// TwinCAT 3 PLC project SPT_PackML_Base
// Title: SPT PackML Base
// Company: Beckhoff Automation LLC
// ProjectVersion: 4.0.0.0
// Description: 4.0.0.0 - Bonkers
// libraries:
//   Intecre.Utilities, * (Intecre Ltd)
//   SPT Event Logger, * (Beckhoff Automation LLC)
//   SPT Utilities, * (Beckhoff Automation LLC)
//   Tc2_Standard, * (Beckhoff Automation GmbH)
//   Tc2_System, * (Beckhoff Automation GmbH)
//   Tc3_EventLogger, * (Beckhoff Automation GmbH)
//   Tc3_Module, * (Beckhoff Automation GmbH)
//   Tc3_PackML_V2, * (Beckhoff Automation GmbH)
//   tcl_SimpleUnitTestLibrary, * (Red Rock Controls Limited)
//   SPT Base Types,newest,Beckhoff Automation LLC
//   SPT Component Base,newest,Beckhoff Automation LLC
// project tree:
//   DUT/ E_PMLUnitMode.TcDUT, ST_PackML_SubUnitInfoExt.TcDUT
//   DUT/HMI/ ST_PackMLBaseModule_Command.TcDUT, ST_PackMLBaseModule_Config.TcDUT, ST_PackMLBaseModule_HMI.TcDUT, ST_PackMLBaseModule_Status.TcDUT
//   Example things/ I_ExampleEquipment.TcIO, T_ExampleModule.TcPOU, T_ExampleMOduleProductionMode.TcPOU
//   / FB_PackML_BaseModule.TcPOU, FB_PackML_ModeLogger.TcPOU, FB_PackML_StateLogger.TcPOU, GlobalTextList.TcGTLO, Parameters_PackML_Base.TcGVL, Task_3.TcTTO, TestUI.TcVIS, Visualization Manager.TcVMO (not stored)
//   Intecre/Axis/ I_Axis.TcIO, I_AxisComponent.TcIO, T_Axis.TcPOU, T_AxisComponent.TcPOU
//   Intecre/CartesianRobot/ I_CartesianRobot.TcIO, I_CartesianRobotModule.TcIO, T_CartesianRobotModule.TcPOU, T_CartesianRobot.TcPOU
//   Intecre/CartesianRobot/Modes/ T_CartesianRobotMaintenanceMode.TcPOU, T_CartesianRobotManualMode.TcPOU, T_CartesianRobotProductionMode.TcPOU
//   Intecre/Collections/ I_ComponentsCollection.TcIO, I_SubModuleCollection.TcIO, T_BaseAlarms.TcPOU, T_CollectionBase.TcPOU, T_ComponentsCollection.TcPOU, T_ExternalControllerCollection.TcPOU, T_SubModuleCollection.TcPOU
//   Intecre/Gripper/ I_Gripper.TcIO, I_GripperModule.TcIO, T_Gripper.TcPOU, T_GripperModule.TcPOU
//   Intecre/Gripper/Modes/ T_GripperMaintenanceMode.TcPOU, T_GripperManualMode.TcPOU, T_GripperProductionMode.TcPOU
//   Intecre/ModeManager/ I_ModeManager.TcIO, T_ModeManager.TcPOU
//   Intecre/PackModes/ I_PackMode.TcIO, I_StateModule.TcIO, T_BaseMode.TcPOU
//   Intecre/Cylinder/ I_Cylinder.TcIO, I_CylinderComponent.TcIO, T_Cylinder.TcPOU, T_CylinderComponent.TcPOU
//   Interfaces/ I_PackML_BaseModule.TcIO, I_PackML_Control.TcIO, I_PackML_ExternalController.TcIO
//   Project Information/ F_GetCompany.TcPOU, F_GetTitle.TcPOU, F_GetVersion.TcPOU
//   Tests/AlarmsTests/ T_BaseAlarmsClearAlarmIfRaisedCleared.TcPOU
//   Tests/CollectionsTests/Components/Mock/ T_ComponentMock.TcPOU (not stored)
//   Tests/CollectionsTests/Components/ T_AddComponentAddedToList.TcPOU, T_AddComponentCompareResultTrue.TcPOU, T_AddMoreThanSizeOfCollectionFalse.TcPOU, T_AddSameComponentTwiceShouldntAdd.TcPOU, T_ClearGroupCountEqualsZeroCompareEqualsFalse.TcPOU, T_ComponentsAllowHmiAllowed.TcPOU, T_ComponentsBlockHmiBlocked.TcPOU (not stored), T_ComponentsIfAnyErrorReturnsErrorTrue.TcPOU (not stored), T_ComponentsInitialisedSuccess.TcPOU (not stored), T_ComponentsResetClearsErrors.TcPOU (not stored), T_CountReturnsCorrect.TcPOU, T_CyclicLogicHasBeenCalledTrue.TcPOU (not stored), T_GetComponentCompareResultsTrue.TcPOU (not stored), T_GetComponentIndexOutOfBoundaryResultsFalse.TcPOU
//   Tests/CollectionsTests/ExternalController/Mock/ T_ExternalControllerMock.TcPOU (not stored)
//   Tests/CollectionsTests/ExternalController/ T_ExternalControllersCollectionNotifyModeChangedSuccess.TcPOU (not stored), T_ExternalControllersCollectionNotifyStateChangedSuccess.TcPOU (not stored)
//   Tests/CollectionsTests/Module/Mock/ T_SubModuleMock.TcPOU (not stored)
//   Tests/CollectionsTests/Module/ T_ModuleCollectionAllInAskedStateReturnsCorrectResponse.TcPOU, T_ModuleCollectionAnyErrorReturnErrorTrue.TcPOU, T_ModuleCollectionAnyInAskedStateReturnsCorrectResponse.TcPOU, T_ModuleCollectionInitialisedSuccess.TcPOU (not stored), T_ModuleCollectionNotifyModeChangedSuccess.TcPOU (not stored), T_ModuleCollectionNotifyStateChangedSuccess.TcPOU (not stored), T_ModuleCollectionOneIsNotInAskedStateReturnsCorrectResponse.TcPOU, T_ModuleCollectionOneNotInitialisedAllNotInitialised.TcPOU, T_ModuleCollectionStateResetReturnsCorrectResponse.TcPOU
//   Tests/ModeAndStateTests/ EquipmentModule.TcPOU, T_CantChangeModInExecute.TcPOU, T_CantChangeStateFromIdleToSuspend.TcPOU, T_JogThroughStates.TcPOU, T_ProductionToMaintenaceInAbort.TcPOU
//   Tests/ModeManagerTests/Mock Objects/ T_MockStateModule.TcPOU
//   Tests/ModeManagerTests/ T_AddCustomPackModeSetsCorrectly.TcPOU, T_AddPackModeSetsCorrectly.TcPOU, T_InitModeManagerWithState.TcPOU, T_ModeChangeFromProductionToMaintenance.TcPOU, T_ModeInitialisedFromInvalidToProduction.TcPOU
//   Tests/ PRG_Tests.TcPOU
//   Version/ Global_Version.TcGVL
//   VISUs/ V_MachineModule.TcVIS, V_Module.TcVIS
// (motion and I/O tree: see PLC project spt_base_types)
// real-time tasks:
//   TASK Task 3: cycle T#10ms, priority 1, ADS port 350

CONFIGURATION SPT_PackML_Base
    RESOURCE PLC ON TwinCAT3
        TASK Task_3(INTERVAL := T#10ms, PRIORITY := 1);
        PROGRAM PRG_Tests WITH Task_3 : PRG_Tests;
    END_RESOURCE
END_CONFIGURATION

// ---- DUT/E_PMLUnitMode.TcDUT
//! @summary Defines the allowable PackML modes  
TYPE E_PMLUnitMode : (
        ePMLUnitMode_Invalid     := 0,
        ePMLUnitMode_Production  := 1,
        ePMLUnitMode_Maintenance := 2,
        ePMLUnitMode_Manual      := 3,
        ePMLUnitMode_UserMode1   := 4,
        ePMLUnitMode_UserMode2   := 5,
        ePMLUnitMode_UserMode3   := 6,
        ePMLUnitMode_UserMode4   := 7,
        ePMLUnitMode_UserMode5   := 8,
        ePMLUnitMode_UserMode6   := 9,
        ePMLUnitMode_UserMode7   := 10,
        ePMLUnitMode_UserMode8   := 11,
        ePMLUnitMode_UserMode9   := 12,
        ePMLUnitMode_UserMode10  := 13,
        ePMLUnitMode_UserMode11  := 14,
        ePMLUnitMode_UserMode12  := 15,
        ePMLUnitMode_UserMode13  := 16,
        ePMLUnitMode_UserMode14  := 17,
        ePMLUnitMode_UserMode15  := 18,
        ePMLUnitMode_UserMode16  := 19,
        ePMLUnitMode_UserMode17  := 20,
        ePMLUnitMode_UserMode18  := 21,
        ePMLUnitMode_UserMode19  := 22,
        ePMLUnitMode_UserMode20  := 23,
        ePMLUnitMode_UserMode21  := 24,
        ePMLUnitMode_UserMode22  := 25,
        ePMLUnitMode_UserMode23  := 26,
        ePMLUnitMode_UserMode24  := 27,
        ePMLUnitMode_UserMode25  := 28,
        ePMLUnitMode_UserMode26  := 29,
        ePMLUnitMode_UserMode27  := 30,
        ePMLUnitMode_UserMode28  := 31
    ) DINT;
END_TYPE

// ---- DUT/HMI/ST_PackMLBaseModule_Command.TcDUT
TYPE ST_PackMLBaseModule_Command :
    STRUCT
        Mode               : E_PMLUnitMode              := Parameters_PackML_Base.UNIT_MODE_DEFAULT;
        State              : Tc3_PackML_V2.E_PMLCommand := Parameters_PackML_Base.UNIT_STATE_DEFAULT;
        ActivateStateLog   : BOOL; //HMI requests to enable the module
        DeactivateStateLog : BOOL; //HMI requests to disable the module
        ActivateModeLog    : BOOL; //HMI requests to enable the module
        DeactivatModeLog   : BOOL; //HMI requests to disable the module
    END_STRUCT
END_TYPE

// ---- DUT/HMI/ST_PackMLBaseModule_Config.TcDUT
TYPE ST_PackMLBaseModule_Config :
    STRUCT
        Name            : STRING;       //Human-readable module name for user-side messaging
        LogStateChanges : BOOL := TRUE; //Toggle to permit or suppress state change logging (Should be tied to HMI setting to optionally reduce event logger clutter)
        LogModeChanges  : BOOL := TRUE; //Toggle to permit or suppress state change logging (Should be tied to HMI setting to optionally reduce event logger clutter)
        ModeNames       : ARRAY[0..31] OF STRING;
    END_STRUCT
END_TYPE

// ---- DUT/HMI/ST_PackMLBaseModule_HMI.TcDUT
TYPE ST_PackMLBaseModule_HMI :
    STRUCT
        Config  : ST_PackMLBaseModule_Config;
        Command : ST_PackMLBaseModule_Command;
        Status  : ST_PackMLBaseModule_Status;
    END_STRUCT
END_TYPE

// ---- DUT/HMI/ST_PackMLBaseModule_Status.TcDUT
TYPE ST_PackMLBaseModule_Status :
    STRUCT
        Busy                : BOOL;
        Error               : BOOL;
        ErrorID             : UDINT;
        Mode                : E_PMLUnitMode;
        State               : Tc3_PackML_V2.E_PMLState;
        HMIControlAvailable : BOOL;
    END_STRUCT
END_TYPE

// ---- DUT/ST_PackML_SubUnitInfoExt.TcDUT
TYPE ST_PackML_SubUnitInfoExt EXTENDS ST_PMLSubUnitInfo : //Extended Struct of ST_PMLSubUnitInfo
    STRUCT
        ModuleID        : DINT;   //Machine ID for messaging and Identification
        ModuleName      : STRING; //Human readable machine name for messaging
        UnitModeCurrent : E_PMLProtectedUnitMode;
        ActiveAlarm     : BOOL;
    END_STRUCT
END_TYPE

// ---- Parameters_PackML_Base.TcGVL
{attribute 'qualified_only'}
VAR_GLOBAL CONSTANT
    MAX_NO_OF_SUBMODULES           : UDINT                       := 20;
    MAX_NO_OF_COMPONENTS           : UDINT                       := 32;
    MAX_NO_OF_EXTERNAL_CONTROLLERS : UDINT                       := 10;
    UNIT_MODE_DEFAULT              : E_PMLUnitMode := E_PMLUnitMode.ePMLUnitMode_Production;
    UNIT_STATE_DEFAULT             : Tc3_PackML_V2.E_PMLCommand  := E_PMLCommand.ePMLCommand_Abort;
	COLLECTION_MAX_SIZE : UDINT := 200;
END_VAR

// ---- Version/Global_Version.TcGVL
{attribute 'TcGenerated'}
{attribute 'no-analysis'}
{attribute 'linkalways'}
// This function has been automatically generated from the project information.
VAR_GLOBAL CONSTANT
	{attribute 'const_non_replaced'}
	stLibVersion_SPT_PackML_Base : ST_LibVersion := (iMajor := 3, iMinor := 0, iBuild := 3, iRevision := 0, nFlags := 1, sVersion := '3.0.3');
END_VAR

// ---- Example things/I_ExampleEquipment.TcIO
INTERFACE I_ExampleEquipment EXTENDS I_PackML_BaseModule

METHOD PUBLIC PickFromStagingArea : BOOL
VAR_INPUT
  orientationOfPick : ST_Orientation;
END_VAR
END_METHOD

END_INTERFACE

// ---- Intecre/Axis/I_Axis.TcIO
INTERFACE I_Axis

END_INTERFACE

// ---- Intecre/Axis/I_AxisComponent.TcIO
INTERFACE I_AxisComponent

END_INTERFACE

// ---- Intecre/CartesianRobot/I_CartesianRobot.TcIO
INTERFACE I_CartesianRobot

METHOD GenericInitialise : BOOL;
VAR_INPUT
	xAxis, yAxis, zAxis : I_Axis;
	gripper : I_Gripper;
END_VAR
END_METHOD

END_INTERFACE

// ---- Intecre/CartesianRobot/I_CartesianRobotModule.TcIO
INTERFACE I_CartesianRobotModule

END_INTERFACE

// ---- Intecre/Collections/I_ComponentsCollection.TcIO
INTERFACE I_ComponentsCollection

END_INTERFACE

// ---- Intecre/Collections/I_SubModuleCollection.TcIO
INTERFACE I_SubModuleCollection

PROPERTY Count : UDINT
GET
END_GET
END_PROPERTY

METHOD TryGetModule: BOOL
VAR_INPUT
	index : UDINT;
END_VAR
VAR_OUTPUT
	Module : I_PackML_BaseModule;
END_VAR
END_METHOD

END_INTERFACE

// ---- Intecre/Gripper/I_Gripper.TcIO
INTERFACE I_Gripper

END_INTERFACE

// ---- Intecre/Gripper/I_GripperModule.TcIO
INTERFACE I_GripperModule

END_INTERFACE

// ---- Intecre/ModeManager/I_ModeManager.TcIO
INTERFACE I_ModeManager

METHOD AddCustomPackMode : BOOL
VAR_INPUT
  index : UINT;
  newPackMode : I_PackMode;
END_VAR
END_METHOD

METHOD AddPackModes : BOOL
VAR_INPUT
  prodMode : I_PackMode;
  maintMode : I_PackMode;
  manMode : I_PackMode;
END_VAR
END_METHOD

METHOD PUBLIC AddStateModule
VAR_INPUT
  stateModule : I_StateModule;
END_VAR
END_METHOD

METHOD PUBLIC ChangeMode
VAR_INPUT
  Mode : E_PMLUnitMode;
END_VAR
END_METHOD

PROPERTY PUBLIC CommandedMode : E_PMLUnitMode
GET
END_GET
END_PROPERTY

PROPERTY CurrentMode : E_PMLUnitMode
GET
END_GET
END_PROPERTY

METHOD PUBLIC CyclicLogic
VAR_INPUT
END_VAR
END_METHOD

PROPERTY PUBLIC LogModeChanges : BOOL
GET
END_GET
SET
END_SET
END_PROPERTY

PROPERTY PUBLIC  ModeNames : REFERENCE TO ARRAY[0..31] OF STRING
GET
END_GET
END_PROPERTY

END_INTERFACE

// ---- Intecre/PackModes/I_PackMode.TcIO
INTERFACE I_PackMode

METHOD Aborted
VAR_INPUT
END_VAR
END_METHOD

METHOD Aborting
VAR_INPUT
END_VAR
END_METHOD

METHOD Clearing
VAR_INPUT
END_VAR
END_METHOD

METHOD Complete
VAR_INPUT
END_VAR
END_METHOD

METHOD Completing
VAR_INPUT
END_VAR
END_METHOD

METHOD Execute
VAR_INPUT
END_VAR
END_METHOD

METHOD Held
VAR_INPUT
END_VAR
END_METHOD

METHOD Holding
VAR_INPUT
END_VAR
END_METHOD

METHOD Idle
VAR_INPUT
END_VAR
END_METHOD

METHOD Resetting
VAR_INPUT
END_VAR
END_METHOD

METHOD Starting
VAR_INPUT
END_VAR
END_METHOD

METHOD Stopped
VAR_INPUT
END_VAR
END_METHOD

METHOD Stopping
VAR_INPUT
END_VAR
END_METHOD

METHOD Suspended
VAR_INPUT
END_VAR
END_METHOD

METHOD Suspending
VAR_INPUT
END_VAR
END_METHOD

METHOD Unholding
VAR_INPUT
END_VAR
END_METHOD

METHOD Unsuspending
VAR_INPUT
END_VAR
END_METHOD

END_INTERFACE

// ---- Intecre/PackModes/I_StateModule.TcIO
INTERFACE I_StateModule

PROPERTY CurrentState : Tc3_PackML_V2.E_PMLState
GET
END_GET
END_PROPERTY

END_INTERFACE

// ---- Intecre/Cylinder/I_Cylinder.TcIO
INTERFACE I_Cylinder

END_INTERFACE

// ---- Intecre/Cylinder/I_CylinderComponent.TcIO
INTERFACE I_CylinderComponent

END_INTERFACE

// ---- Interfaces/I_PackML_BaseModule.TcIO
INTERFACE I_PackML_BaseModule EXTENDS I_CyclicFB, I_PackML_Control

PROPERTY CurrentAlarmSeverity : TcEventSeverity
GET
END_GET
END_PROPERTY

PROPERTY LogModeChanges : BOOL
GET
END_GET
SET
END_SET
END_PROPERTY

PROPERTY LogStateChanges : BOOL
GET
END_GET
SET
END_SET
END_PROPERTY

PROPERTY Name : STRING
GET
END_GET
SET
END_SET
END_PROPERTY

PROPERTY ParentResponseDefinitions : ARRAY[0..4] OF E_AlarmResponse
GET
END_GET
SET
END_SET
END_PROPERTY

END_INTERFACE

// ---- Interfaces/I_PackML_Control.TcIO
INTERFACE I_PackML_Control EXTENDS I_InterfaceBase

METHOD ChangeMode
VAR_INPUT
    Mode : E_PMLUnitMode;
END_VAR
END_METHOD

METHOD ChangeState
VAR_INPUT
    State : E_PMLCommand;
END_VAR
END_METHOD

PROPERTY CurrentMode : E_PMLUnitMode
GET
END_GET
END_PROPERTY

PROPERTY CurrentState : E_PMLState
GET
END_GET
END_PROPERTY

PROPERTY ModeCommand : DINT
GET
END_GET
SET
END_SET
END_PROPERTY

PROPERTY StateCommand : E_PMLCommand
GET
END_GET
SET
END_SET
END_PROPERTY

END_INTERFACE

// ---- Interfaces/I_PackML_ExternalController.TcIO
INTERFACE I_PackML_ExternalController EXTENDS I_InterfaceBase

PROPERTY Control : I_PackML_Control
SET
END_SET
END_PROPERTY

METHOD ModeChanged
VAR_INPUT
    NewMode : E_PMLUnitMode;
END_VAR
END_METHOD

METHOD StateChanged
VAR_INPUT
    NewState : E_PMLCommand;
END_VAR
END_METHOD

END_INTERFACE

// ---- Tests/PRG_Tests.TcPOU
PROGRAM PRG_Tests
VAR
  testRunner : T_TestRunner;
  
  //Modes
  modeTestSuite : T_TestSuite;
  ProductionToMaintenaceInAbort : T_ProductionToMaintenaceInAbort(modeTestSuite);
  CantChangeModInExecute : T_CantChangeModInExecute(modeTestSuite);
  JogThroughStates : T_JogThroughStates(modeTestSuite);
  CantChangeStateFromIdleToSuspend : T_CantChangeStateFromIdleToSuspend(modeTestSuite);
  
  // set mode
  AddPackModeSetsCorrectly : T_AddPackModeSetsCorrectly(modeTestSuite);  
  InitModeManagerWithState : T_InitModeManagerWithState(modeTestSuite);
  ModeChangeFromProductionToMaintenance : T_ModeChangeFromProductionToMaintenance(modeTestSuite);
  ModeInitialisedFromInvalidToProduction : T_ModeInitialisedFromInvalidToProduction(modeTestSuite);
  AddCustomPackModeSetsCorrectly : T_AddCustomPackModeSetsCorrectly(modeTestSuite);
  
    //collections tests
  CollectionsTestSuite : T_TestSuite;
  AddComponentAddedToList : T_AddComponentAddedToList (CollectionsTestSuite);
  AddComponentCompareResultTrue : T_AddComponentCompareResultTrue(CollectionsTestSuite);
  CountReturnsCorrect : T_CountReturnsCorrect(CollectionsTestSuite);
  GetComponentCompareResultsTrue : T_GetComponentCompareResultsTrue(CollectionsTestSuite);
  ClearGroupCountEqualsZeroCompareEqualsFalse : T_ClearGroupCountEqualsZeroCompareEqualsFalse(CollectionsTestSuite);
  AddSameComponentTwiceShouldntAdd : T_AddSameComponentTwiceShouldntAdd(CollectionsTestSuite);
  GetComponentIndexOutOfBoundaryResultsFalse : T_GetComponentIndexOutOfBoundaryResultsFalse(CollectionsTestSuite);
  AddMoreThanSizeOfCollectionFalse : T_AddMoreThanSizeOfCollectionFalse(CollectionsTestSuite);
  CyclicLogicHasBeenCalledTrue : T_CyclicLogicHasBeenCalledTrue(CollectionsTestSuite);
  ComponentsInitialisedSuccess : T_ComponentsInitialisedSuccess (CollectionsTestSuite);
  ComponentsIfAnyErrorReturnsErrorTrue : T_ComponentsIfAnyErrorReturnsErrorTrue (CollectionsTestSuite);
  ComponentsAllowHmiAllowed : T_ComponentsAllowHmiAllowed (CollectionsTestSuite);
  ComponentsBlockHmiBlocked : T_ComponentsBlockHmiBlocked (CollectionsTestSuite);
  ComponentsResetClearsErrors : T_ComponentsResetClearsErrors (CollectionsTestSuite);
  ExternalControllersCollectionNotifyStateChangedSuccess : T_ExternalControllersCollectionNotifyStateChangedSuccess (CollectionsTestSuite);
  ExternalControllersCollectionNotifyModeChangedSuccess : T_ExternalControllersCollectionNotifyModeChangedSuccess (CollectionsTestSuite);
  ModuleCollectionNotifyModeChangedSuccess : T_ModuleCollectionNotifyModeChangedSuccess (CollectionsTestSuite);
  ModuleCollectionNotifyStateChangedSuccess : T_ModuleCollectionNotifyStateChangedSuccess (CollectionsTestSuite);
  ModuleCollectionInitialisedSuccess : T_ModuleCollectionInitialisedSuccess (CollectionsTestSuite);
  ModuleCollectionOneNotInitialisedAllNotInitialised : T_ModuleCollectionOneNotInitialisedAllNotInitialised (CollectionsTestSuite);
  ModuleCollectionAnyErrorReturnErrorTrue : T_ModuleCollectionAnyErrorReturnErrorTrue (CollectionsTestSuite);
  ModuleCollectionAllInAskedStateReturnsCorrectResponse : T_ModuleCollectionAllInAskedStateReturnsCorrectResponse (CollectionsTestSuite);
  ModuleCollectionOneIsNotInAskedStateReturnsCorrectResponse : T_ModuleCollectionOneIsNotInAskedStateReturnsCorrectResponse (CollectionsTestSuite);
  ModuleCollectionAnyInAskedStateReturnsCorrectResponse : T_ModuleCollectionAnyInAskedStateReturnsCorrectResponse (CollectionsTestSuite);
  ModuleCollectionStateResetReturnsCorrectResponse : T_ModuleCollectionStateResetReturnsCorrectResponse (CollectionsTestSuite);
END_VAR

IF testRunner.ReloadTests THEN
    testRunner.AddTestSuite(modeTestSuite);
    testRunner.AddTestSuite(CollectionsTestSuite);
    testRunner.ReloadTests := FALSE;
END_IF

testRunner();

END_PROGRAM

// ---- Tests/ModeAndStateTests/T_ProductionToMaintenaceInAbort.TcPOU
FUNCTION_BLOCK T_ProductionToMaintenaceInAbort EXTENDS T_UnitTestBase
VAR
  em : EquipmentModule; 
  actual, expected : E_PMLUnitMode;
  scanCounter: INT;
  cmdTriggered : BOOL;
  myTestState : (ARRANGE, ACT, ASSERT);
END_VAR

CASE myTestState OF

  ARRANGE:
    em.CyclicLogic();

    IF em.InitComplete THEN
      myTestState := ACT;
      CycleModuleLogicToAllowChangesToFilterThrough();
    END_IF

  ACT:

    CycleModuleLogicToAllowChangesToFilterThrough();
    em.ChangeMode(E_PMLUnitMode.ePMLUnitMode_Maintenance);
    CycleModuleLogicToAllowChangesToFilterThrough();
    actual := em.CurrentMode;
    expected := E_PMLUnitMode.ePMLUnitMode_Maintenance;
    myTestState := ASSERT;

  ASSERT:

    assertion.AssertEquals_UINT(TO_UINT(actual), TO_UINT(expected), 'actual := equipmentModule.CurrentMode');
    myTestState := ARRANGE;
    cmdTriggered := FALSE;
    TestFinished();

END_CASE

METHOD CycleModuleLogicToAllowChangesToFilterThrough : BOOL
VAR_INST
	i: INT;

END_VAR
//em.CyclicLogic();
//CycleModuleLogicToAllowChangesToFilterThrough := i >= 10;
//i := SEL(i >= 10, i + 1, 0);

FOR i := 0 TO 10 DO
  em.CyclicLogic();
END_FOR
END_METHOD

END_FUNCTION_BLOCK

// ---- Tests/ModeAndStateTests/EquipmentModule.TcPOU
FUNCTION_BLOCK EquipmentModule EXTENDS FB_PackML_BaseModule
VAR_INPUT
END_VAR
VAR_OUTPUT
END_VAR
VAR
END_VAR

END_FUNCTION_BLOCK

// ---- FB_PackML_BaseModule.TcPOU
FUNCTION_BLOCK ABSTRACT FB_PackML_BaseModule EXTENDS FB_CyclicFB IMPLEMENTS I_PackML_BaseModule, I_PackML_Control, I_StateModule
  //I_PMLControl
VAR

  _CurrentState : Tc3_PackML_V2.E_PMLState;
  _CommandedState : Tc3_PackML_V2.E_PMLCommand;
END_VAR

VAR
  _CurrentAlarmSeverity : TcEventSeverity;
  _LogStateChanges : BOOL := FALSE; //Toggle to permit or suppress state change logging (Should be tied to HMI setting to optionally reduce event logger clutter)
  _Name : STRING; //Human-readable module name for user-side messaging
  _ParentFaultResponseDefinitions : ARRAY[0..4] OF E_AlarmResponse
    := [E_AlarmResponse.NoResponse,
    E_AlarmResponse.NoResponse, E_AlarmResponse.NoResponse, E_AlarmResponse.Abort_ImmediateError, E_AlarmResponse.Abort_ImmediateError];
END_VAR

VAR

  ModeManager : T_ModeManager(THIS^);
  InitialiseStates : (init,
    CountSubModules,
    SetSizeOfArrays,
    WaitForInitializeComplete);
  ComponentsCollection : T_ComponentsCollection;
  SubModulesCollection : T_SubModuleCollection;
  ExternalControllersCollection : T_ExternalControllerCollection;
  BaseAlarms : T_BaseAlarms;

  //spt classes    
  StateMachine : PML_StateMachine; //Manages PackML state transitions   
  PrevState : Tc3_PackML_V2.E_PMLState; //Last cycle PackML state 
  PMLStateLogger : FB_PackML_StateLogger; //Logs PackML state changes

  PackMLAlarms : ARRAY[1..48] OF FB_TcAlarm; //Array of alarms for PackML state and mode changes that exist in any PackML enabled module
  ipSubModules : ARRAY[1..Parameters_PackML_Base.MAX_NO_OF_SUBMODULES] OF I_PackML_BaseModule;
  NumberOfSubModules : UDINT := 0; //calculated number of instantiated sub modules
  ReachedInitialDefaultStateAndMode : BOOL;

  HMICommand_RT : R_TRIG;
  HMICommandActive_Base : BOOL;
  HMICommandActive_Descendant : BOOL;
  PackMLBaseModule_HMI : ST_PackMLBaseModule_HMI; //Handles status and control communications with the HMI
END_VAR

//*********************************************************

// !!!!! Code implementation only in CyclicLogic() method !!!!! 

//*********************************************************

//! @summary This method contains code which will execute when this PackML module is in the <b>Aborted</b> state
METHOD PROTECTED Aborted

(*! <description> <b>The base implementation of this method is empty. User must override this method to provide functionality.</b>
<table> 
	<tr>
		<th> Previous State </th>
		<th> Transition In </th>
		<th> Transition Out </th>
		<th> Next State  </th> 
	</tr>
	<tr>
		<td> Aborting </td>
		<td> State Complete <i>(Aborting)</i></td> 
		<td> Clear Command </td>
		<td> Clearing </td> 
	</tr>
</table>
This method is called as required by <c>StateControl()</c>
</description> 

*)
//*************************************************************************************************************************************************************************

//If you are about to write application specific code, note that any such code should exist within the "Application" directory using a Function Block that 'EXTENDS' this base Function Block!

//This particular method's functionality can be overriden in the extended block by creating a method of the same name, with desired functionality therein

//If the functionality of this base module is to be retained, but more functionality is desired, the extended method can contain a SUPER^.ThisMethodName(); call, which will call this code

//*************************************************************************************************************************************************************************
END_METHOD

//! @summary Provides fault reaction logic where the module state is driven to the <b>Aborting</b> state
METHOD PROTECTED AbortImmediate

//! @description No error is thrown by this fault reaction.

//! @description This method is called by <c>ComponentMonitor()</c> or <c>SubModuleMonitor()</c> as required
ChangeState(E_PMLCommand.ePMLCommand_Abort);
END_METHOD

//! @summary Provides fault reaction logic where the module state is driven to the <b>Aborting</b> state
METHOD PROTECTED AbortImmediateError
VAR_INPUT
    Name     : STRING; //! The name of the faulting submodule or component
    IsModule : BOOL;   //! If TRUE a SubModuleError is thrown.  If FALSE a ComponentError is thrown. 
END_VAR

//! @description This fault reaction throws an accompanying error

//! @description This method is called by <c>ComponentMonitor()</c> or <c>SubModuleMonitor()</c> as required
//IF IsModule THEN
//    IF NOT BaseAlarms[E_BaseAlarms.SubModuleError].bRaised THEN
//        F_RaiseAlarmWithStringParameters(BaseAlarms[E_BaseAlarms.SubModuleError],
//                                         _Name,
//                                         '',
//                                         '');
//    END_IF
//ELSE
//    IF NOT BaseAlarms[E_BaseAlarms.ComponentError].bRaised THEN
//        F_RaiseAlarmWithStringParameters(BaseAlarms[E_BaseAlarms.ComponentError],
//                                         _Name,
//                                         '',
//                                         '');
//    END_IF
//END_IF

IF IsModule THEN
	BaseAlarms.RaiseAlarmWithStringParameters(E_BaseAlarms.SubModuleError, _name, '','');
ELSE
	BaseAlarms.RaiseAlarmWithStringParameters(E_BaseAlarms.ComponentError, _name, '','');
END_IF

THIS^.ChangeState(E_PMLCommand.ePMLCommand_Abort);
END_METHOD

//! @summary This method contains code which will execute when this PackML module is in the <b>Aborting</b> state
METHOD PROTECTED Aborting
(*! <description> <b>Note:</b> The <i>Abort</i> command should be associated with the fault handing routine of a module. It should not be directly commanded from any user inteface. 

<table> 
	<tr>
		<th> Previous State </th>
		<th> Transition In </th>
		<th> Transition Out </th>
		<th> Next State  </th> 
	</tr>
	<tr>
		<td> <b>ANY</b> </td>
		<td> Abort Command </td> 
		<td> State Complete </td>
		<td> Aborted </td> 
	</tr>
</table>

This method is called as required by <c>StateControl()</c>
</description> 

*)
//*************************************************************************************************************************************************************************

//If you are about to write application specific code, note that any such code should exist within the "Application" directory using a Function Block that 'EXTENDS' this base Function Block!

//This particular method's functionality can be overriden in the extended block by creating a method of the same name, with desired functionality therein

//If the functionality of this base module is to be retained, but more functionality is desired, the extended method can contain a SUPER^.ThisMethodName(); call, which will call this code

//*************************************************************************************************************************************************************************

//Perform State tasks here

// Send abort command to all sub modules
SubModulesCollection.NotifyStateChanged(ePMLCommand_Abort);

IF NOT SubModulesCollection.AllInRequestedState(ePMLState_Aborted) THEN
	RETURN;
END_IF

StateComplete();
END_METHOD

//! @summary Sets permissive bit to allow HMI control of module and component functions
METHOD PROTECTED FINAL AllowHMIControl
VAR_INPUT
    ThisModuleOnly : BOOL; //! If TRUE, only the PackML module itself is controllable. If FALSE, all components become controllable as well
END_VAR

VAR
    i : UDINT;
END_VAR

//! @description This method is called as required by the <c>HMIPermissions()</c> method
PackMLBaseModule_HMI.Status.HMIControlAvailable := TRUE;
IF ThisModuleOnly THEN
	componentsCollection.BlockHmiControl();	
ELSE
	componentsCollection.AllowHMIControl();
END_IF
END_METHOD

//! @summary Clears permissive bit to disallow HMI control of module and component functions
METHOD PROTECTED FINAL BlockHMIControl
VAR
    i : UDINT;
END_VAR

//! @description This method is called as required by the <c>HMIPermissions()</c> method
PackMLBaseModule_HMI.Status.HMIControlAvailable := FALSE;
componentsCollection.BlockHMIControl();
END_METHOD

METHOD ChangeMode
VAR_INPUT
    Mode : E_PMLUnitMode;
END_VAR
ModeManager.ChangeMode(Mode);
PackMLBaseModule_HMI.Command.Mode := Mode;
ExternalControllersCollection.NotifyModeChanged(Mode);
END_METHOD

METHOD ChangeState
VAR_INPUT
    State : E_PMLCommand;
END_VAR
IF State <> _CommandedState THEN
    StateCommand := State;
END_IF
END_METHOD

//! @summary This method contains code which will execute when this PackML module is in the <b>Clearing</b> state
METHOD PROTECTED Clearing
VAR
    i               : UDINT;
    SubModulesReady : BOOL := TRUE;
END_VAR

(*! <description> <b>Note:</b> The <i>Clear</i> command can also be thought of as a <i>fault reset</i> depite the ambiguity in the naming of the <i>Reset</i> state. 
<table> 
	<tr>
		<th> Previous State </th>
		<th> Transition In </th>
		<th> Transition Out </th>
		<th> Next State  </th> 
	</tr>
	<tr>
		<td> Aborted </td>
		<td> Clear Command </td> 
		<td> State Complete </td>
		<td> Stopped </td> 
	</tr>
</table>
This method is called as required by <c>StateControl()</c>
</description> 

*)
//*************************************************************************************************************************************************************************

//If you are about to write application specific code, note that any such code should exist within the "Application" directory using a Function Block that 'EXTENDS' this base Function Block!

//This particular method's functionality can be overriden in the extended block by creating a method of the same name, with desired functionality therein

//If the functionality of this base module is to be retained, but more functionality is desired, the extended method can contain a SUPER^.ThisMethodName(); call, which will call this code

//*************************************************************************************************************************************************************************

//Perform State tasks here

// Send clear command to all sub modules

SubModulesCollection.NotifyStateChanged(ePMLCommand_Clear);

baseAlarms.ClearAlarmIfRaised(E_BaseAlarms.ComponentError, resetConfirmation:= FALSE);
baseAlarms.ClearAlarmIfRaised(E_BaseAlarms.SubModuleError, resetConfirmation:= FALSE);

//IF BaseAlarms[E_BaseAlarms.ComponentError].bRaised THEN
//    BaseAlarms[E_BaseAlarms.ComponentError].Clear(0, FALSE);
//END_IF;

//IF BaseAlarms[E_BaseAlarms.SubModuleError].bRaised THEN
//    BaseAlarms[E_BaseAlarms.SubModuleError].Clear(0, 0);
//END_IF;

componentsCollection.Reset();
IF NOT SubModulesCollection.AllInRequestedState(ePMLState_Stopped) OR componentsCollection.AnyError THEN
 	RETURN;
END_IF

StateComplete();
END_METHOD

//! @summary This method contains code which will execute when this PackML module is in the <b>Complete</b> state
METHOD PROTECTED Complete

(*! <description> <b>The base implementation of this method is empty. User must override this method to provide functionality.</b>
<table> 
	<tr>
		<th> Previous State </th>
		<th> Transition In </th>
		<th> Transition Out </th>
		<th> Next State  </th> 
	</tr>
	<tr>
		<td> Completing </td>
		<td> State Complete <i>(Completing)</i></td> 
		<td> Reset Command </td>
		<td> Resetting </td> 
	</tr>
</table>
This method is called as required by <c>StateControl()</c>
</description> 

*)
//*************************************************************************************************************************************************************************

//If you are about to write application specific code, note that any such code should exist within the "Application" directory using a Function Block that 'EXTENDS' this base Function Block!

//This particular method's functionality can be overriden in the extended block by creating a method of the same name, with desired functionality therein

//If the functionality of this base module is to be retained, but more functionality is desired, the extended method can contain a SUPER^.ThisMethodName(); call, which will call this code

//*************************************************************************************************************************************************************************
END_METHOD

//! @summary This method contains code which will execute when this PackML module is in the <b>Completing</b> state
METHOD PROTECTED Completing

(*! <description><b></b><table> 
	<tr>
		<th> Previous State </th>
		<th> Transition In </th>
		<th> Transition Out </th>
		<th> Next State  </th> 
	</tr>
	<tr>
		<td> Execute </td>
		<td> State Complete <i>(Execute)</i> </td> 
		<td> State Complete </td>
		<td> Completed </td> 
	</tr>
</table>
This method is called as required by <c>StateControl()</c>
</description> 
*)
//*************************************************************************************************************************************************************************

//If you are about to write application specific code, note that any such code should exist within the "Application" directory using a Function Block that 'EXTENDS' this base Function Block!

//This particular method's functionality can be overriden in the extended block by creating a method of the same name, with desired functionality therein

//If the functionality of this base module is to be retained, but more functionality is desired, the extended method can contain a SUPER^.ThisMethodName(); call, which will call this code

//*************************************************************************************************************************************************************************

//Perform State tasks here

// Send complete command to all sub modules
SubModulesCollection.NotifyStateChanged(ePMLCommand_Complete);

IF NOT SubModulesCollection.AllInRequestedState(ePMLState_Complete) THEN
	RETURN;
END_IF

StateComplete();
END_METHOD

//! @summary This method monitors <b>components</b> within this PackML module and initiates fault responses as required
METHOD PROTECTED ComponentMonitor : BOOL
VAR
    AlarmResponses : ARRAY[0..4] OF SPT_ComponentBase.E_AlarmResponse; //Temporary response array
    i              : UDINT;
	
END_VAR

//! @description This method is called cyclically by <c>CyclicLogic()</c>
//TODO handle this with collection 



//FOR i := 1 TO NumberOfComponents DO
//    IF _CurrentState <> E_PMLState.ePMLState_Aborted AND _CurrentState <> E_PMLState.ePMLState_Aborting AND _CurrentState <> E_PMLState.ePMLState_Clearing AND
//       _CurrentState <> E_PMLState.ePMLState_Stopped AND _CurrentState <> E_PMLState.ePMLState_Stopping THEN
//        AlarmResponses := ipComponents[i].ParentResponseDefinitions;
//        CASE AlarmResponses[ipComponents[i].CurrentAlarmSeverity] OF
//            E_AlarmResponse.Abort_ImmediateError:
//                AbortImmediateError(ipComponents[i].Name, FALSE);

//            E_AlarmResponse.Abort_Immediate:
//                AbortImmediate();

//            E_AlarmResponse.Stop_Immediate:
//                StopImmediate();

//            E_AlarmResponse.Stop_Controlled:
//                StopControlled();

//            E_AlarmResponse.Hold_Immediate:
//                HoldImmediate();

//            E_AlarmResponse.Suspend_Immediate:
//                SuspendImmediate();

//            E_AlarmResponse.Suspend_Controlled:
//                SuspendControlled();

//            E_AlarmResponse.NoResponse:
//                ;
//        END_CASE
//    ELSIF _CurrentState = E_PMLState.ePMLState_Stopped OR _CurrentState = E_PMLState.ePMLState_Stopping THEN
//        AlarmResponses := ipComponents[i].ParentResponseDefinitions;
//        CASE AlarmResponses[ipComponents[i].CurrentAlarmSeverity] OF
//            E_AlarmResponse.Abort_ImmediateError:
//                AbortImmediateError(ipComponents[i].Name, FALSE);

//            E_AlarmResponse.Abort_Immediate:
//                AbortImmediate();

//            E_AlarmResponse.NoResponse:
//                ;
//        END_CASE
//    END_IF
//END_FOR
END_METHOD

//! @summary Initializes event function blocks using this module's name
{attribute 'call_after_online_change_slot' := '<slot>'}
METHOD PROTECTED CreateEvents

//! @description This method is called by <c>Initialize()</c> as required
F_CreateAllEventsInClass(Alarms     := PackMLAlarms,
                         ClassSize  := SIZEOF(TC_EVENTS.PackMLBase_Alarms),
                         pInitEvent := ADR(TC_EVENTS.PackMLBase_Alarms.InitReferenceEvent),
                         Prefix     := _Name);

F_CreateAllEventsInClass(Alarms     := BaseAlarms.AlarmsArray,
                         ClassSize  := SIZEOF(TC_EVENTS.BaseAlarms),
                         pInitEvent := ADR(TC_EVENTS.BaseAlarms.InitReferenceEvent),
                         Prefix     := _Name);
END_METHOD

//! @summary Returns the highest severity of any event(s) currently raised 
PROPERTY CurrentAlarmSeverity : TcEventSeverity
GET
CurrentAlarmSeverity := _CurrentAlarmSeverity;
END_GET
END_PROPERTY

PROPERTY CurrentMode : E_PMLUnitMode
GET
CurrentMode := ModeManager.CurrentMode;
END_GET
END_PROPERTY

//! @summary Returns current PackML state of this module
PROPERTY CurrentState : Tc3_PackML_V2.E_PMLState
GET
CurrentState := _CurrentState;
END_GET
END_PROPERTY

//! @summary This method serves as the entry point for all underlying FB logic

//! @description This method should be called cyclically by descendant function blocks by invoking <c>SUPER^.CyclicLogic()</c>.  Alternatively, the contents of this method could be reimplemented entirely in which case a call to this method would not be necessary.
METHOD PUBLIC CyclicLogic
VAR
    i : UDINT;
END_VAR
//*********************************************************

//If you are about to write actual machine implementation code, note that implementation code should exist within an implementation machine module block that extends this machine module base!

//*********************************************************

// Descendents of this FB which override this methods should

// use SUPER^.Initialize()
IF NOT _InitComplete THEN
    _InitComplete := Initialize();
    RETURN;
END_IF

// Inhibit mode & state errors until startup is complete
IF NOT ReachedInitialDefaultStateAndMode AND _CurrentState = E_PMLState.ePMLState_Aborted AND ModeManager.CurrentMode = Parameters_PackML_Base.UNIT_MODE_DEFAULT THEN
    ReachedInitialDefaultStateAndMode := TRUE;
END_IF

// Call this module's subunits, if any are defined
SubModulesCollection.CyclicLogic();
//SubModulesCollection.SetSubModuleInfoState(PMLSubModuleInfo);

componentsCollection.CyclicLogic();

//Handle HMI communications--this must happen before state control!!
HMICommunication();

// Mode control loop of the module
ModeManager.CyclicLogic();
//ModeControl();

// State control loop of the module
StateControl();

//VISUCommunication();

//ExternalControl();
SubModuleMonitor();
ComponentMonitor();
HMIPermissions();
_CurrentAlarmSeverity := TcEventSeverity.Verbose;
_CurrentAlarmSeverity := F_GetMaxSeverityRaised(Alarms := PackMLAlarms, CurrentSeverity := _CurrentAlarmSeverity);
_CurrentAlarmSeverity := F_GetMaxSeverityRaised(Alarms := BaseAlarms.AlarmsArray, CurrentSeverity := _CurrentAlarmSeverity);
END_METHOD

//! @summary This method contains code which will execute when this PackML module is in the <b>Execute</b> state
METHOD PROTECTED Execute

(*! <description> <b>The base implementation of this method is empty. User must override this method to provide functionality.</b>
<table> 
	<tr>
		<th> Previous State </th>
		<th> Transition In </th>
		<th> Transition Out </th>
		<th> Next State  </th> 
	</tr>
	<tr>
		<td> Starting<b>-or-</b>Unholding <b>-or-</b>Unsuspending</td>
		<td> State Complete<i>(Starting<b>-or-</b>Unholding<b>-or-</b>Unsuspending)</i></td> 
		<td> State Complete<b>-or-</b>Hold Command<b>-or-</b>Suspend Command</td>
		<td> Completing<b>-or-</b>Holding<b>-or-</b>Suspending</td>
	</tr>
</table>
This method is called as required by <c>StateControl()</c>
</description> 

*)
//*************************************************************************************************************************************************************************

//If you are about to write application specific code, note that any such code should exist within the "Application" directory using a Function Block that 'EXTENDS' this base Function Block!

//This particular method's functionality can be overriden in the extended block by creating a method of the same name, with desired functionality therein

//If the functionality of this base module is to be retained, but more functionality is desired, the extended method can contain a SUPER^.ThisMethodName(); call, which will call this code

//*************************************************************************************************************************************************************************

ModeManager.CurrentStrategy.Execute();
END_METHOD

//! @summary This method contains code which will execute when this PackML module is in the <b>Held</b> state
METHOD PROTECTED Held

(*! <description> <b>The base implementation of this method is empty. User must override this method to provide functionality.</b>
<table> 
	<tr>
		<th> Previous State </th>
		<th> Transition In </th>
		<th> Transition Out </th>
		<th> Next State  </th> 
	</tr>
	<tr>
		<td> Holding </td>
		<td> State Complete <i>(Holding)</i></td> 
		<td> Unhold Command </td>
		<td> Unholding </td> 
	</tr>
</table>
This method is called as required by <c>StateControl()</c>
</description> 

*)
//*************************************************************************************************************************************************************************

//If you are about to write application specific code, note that any such code should exist within the "Application" directory using a Function Block that 'EXTENDS' this base Function Block!

//This particular method's functionality can be overriden in the extended block by creating a method of the same name, with desired functionality therein

//If the functionality of this base module is to be retained, but more functionality is desired, the extended method can contain a SUPER^.ThisMethodName(); call, which will call this code

//*************************************************************************************************************************************************************************
END_METHOD

//! @summary Provides interlocks for HMI control and updates HMI status information for this module
METHOD PROTECTED HMICommunication

//! @description This method is called cyclically by <c>CyclicLogic()</c>
//Extend this method in extended FBs to communicate specific implementation data

//Process HMI requests
HMICommand_RT(CLK := (PackMLBaseModule_HMI.Status.HMIControlAvailable AND NOT HMICommandActive_Descendant) AND
                     (PackMLBaseModule_HMI.Command.ActivateModeLog XOR PackMLBaseModule_HMI.Command.DeactivatModeLog XOR PackMLBaseModule_HMI.Command.ActivateStateLog XOR
                     PackMLBaseModule_HMI.Command.DeactivateStateLog XOR PackMLBaseModule_HMI.Command.Mode <> ModeManager.CommandedMode XOR PackMLBaseModule_HMI.Command.State <> _CommandedState));

//Desendant components should observe this to interlock HMI commands
HMICommandActive_Base := PackMLBaseModule_HMI.Status.HMIControlAvailable AND
                         (PackMLBaseModule_HMI.Command.ActivateModeLog OR PackMLBaseModule_HMI.Command.DeactivatModeLog OR PackMLBaseModule_HMI.Command.ActivateStateLog OR
                         PackMLBaseModule_HMI.Command.DeactivateStateLog XOR PackMLBaseModule_HMI.Command.Mode <> ModeManager.CommandedMode XOR PackMLBaseModule_HMI.Command.State <> _CommandedState);

IF HMICommand_RT.Q THEN
    IF PackMLBaseModule_HMI.Command.ActivateModeLog THEN
        ModeManager.LogModeChanges := TRUE;
    END_IF

    IF PackMLBaseModule_HMI.Command.DeactivatModeLog THEN
        ModeManager.LogModeChanges := FALSE;
    END_IF

    IF PackMLBaseModule_HMI.Command.ActivateStateLog THEN
        LogStateChanges := TRUE;
    END_IF

    IF PackMLBaseModule_HMI.Command.DeactivateStateLog THEN
        _LogStateChanges := FALSE;
    END_IF

    IF PackMLBaseModule_HMI.Command.Mode <> ModeManager.CommandedMode THEN
        ModeCommand := PackMLBaseModule_HMI.Command.Mode;
    END_IF

    IF PackMLBaseModule_HMI.Command.State <> _CommandedState THEN
        StateCommand := PackMLBaseModule_HMI.Command.State;
    END_IF
END_IF

PackMLBaseModule_HMI.Config.Name            := _Name;
PackMLBaseModule_HMI.Config.LogModeChanges  := ModeManager.LogModeChanges;
PackMLBaseModule_HMI.Config.LogStateChanges := _LogStateChanges;
PackMLBaseModule_HMI.Config.ModeNames       := ModeManager.ModeNames;
PackMLBaseModule_HMI.Status.Mode            := ModeManager.CurrentMode;
PackMLBaseModule_HMI.Status.State           := _CurrentState;
PackMLBaseModule_HMI.Status.Busy            := _Busy;
PackMLBaseModule_HMI.Status.Error           := _Error;
PackMLBaseModule_HMI.Status.ErrorID         := _ErrorID;
END_METHOD

//! @summary Automatically enables and disables HMI control based on the PackML mode
METHOD PROTECTED HMIPermissions

//! @description This method is called cyclically by <c>CyclicLogic()</c>
//General Mode Based Monitoring and handling of HMI control
CASE ModeManager.CurrentMode OF
    E_PMLUnitMode.ePMLUnitMode_Production:
        CASE _CurrentState OF
            E_PMLState.ePMLState_Stopped:
                AllowHMIControl(ThisModuleOnly := TRUE); //Allow control for recovery
            E_PMLState.ePMLState_Idle:
                BlockHMIControl();
            E_PMLState.ePMLState_Suspended:
                BlockHMIControl();
            E_PMLState.ePMLState_Execute:
                BlockHMIControl();
            E_PMLState.ePMLState_Aborted:
                AllowHMIControl(ThisModuleOnly := TRUE); //Allow control for recovery
            E_PMLState.ePMLState_Held:
                AllowHMIControl(ThisModuleOnly := TRUE); //Allow control for recovery
            E_PMLState.ePMLState_Complete:
                BlockHMIControl();
        END_CASE
    E_PMLUnitMode.ePMLUnitMode_Manual:
        AllowHMIControl(ThisModuleOnly := FALSE);
    E_PMLUnitMode.ePMLUnitMode_Maintenance:
        AllowHMIControl(ThisModuleOnly := FALSE);
END_CASE
END_METHOD

//! @summary Provides fault reaction logic where the module state is driven to the <b>Holding</b> state at the next available opportunity
METHOD PROTECTED HoldControlled

(*! <description> No error is thrown by this fault reaction.
	<b> TODO: Needs implementation </b> </description>*)

//! @description This method is called by <c>ComponentMonitor()</c> or <c>SubModuleMonitor()</c> as required
ChangeState(E_PMLCommand.ePMLCommand_Hold);
END_METHOD

//! @summary Provides fault reaction logic where the module state is driven to the <b>Holding</b> state immediately
METHOD PROTECTED HoldImmediate

(*! <description> No error is thrown by this fault reaction.
	<b> TODO: Needs implementation </b> </description>*)

//! @description This method is called by <c>ComponentMonitor()</c> or <c>SubModuleMonitor()</c> as required
ChangeState(E_PMLCommand.ePMLCommand_Hold);
END_METHOD

//! @summary This method contains code which will execute when this PackML module is in the <b>Holding</b> state
METHOD PROTECTED Holding
VAR
    i               : UDINT;
    SubModulesReady : BOOL := TRUE;
END_VAR

(*! <description><b>Note:</b> The <i>Hold</i> command is intended to be given by an operator. It is meant to be distinct from a <i>Suspend</i> in that upstream/downstream jams, etc. should be handled automatically using <i>Suspend</i>.  Both <i>Hold</i>and<i>Suspend</i> result in a <i>paused</i> state which should allow resumption of the <b>Execute</b> state. 
<table> 
	<tr>
		<th> Previous State </th>
		<th> Transition In </th>
		<th> Transition Out </th>
		<th> Next State  </th> 
	</tr>
	<tr>
		<td> Execute </td>
		<td> Hold Command </td> 
		<td> State Complete </td>
		<td> Held </td> 
	</tr>
</table>
This method is called as required by <c>StateControl()</c>
</description> 

*)
//*************************************************************************************************************************************************************************

//If you are about to write application specific code, note that any such code should exist within the "Application" directory using a Function Block that 'EXTENDS' this base Function Block!

//This particular method's functionality can be overriden in the extended block by creating a method of the same name, with desired functionality therein

//If the functionality of this base module is to be retained, but more functionality is desired, the extended method can contain a SUPER^.ThisMethodName(); call, which will call this code

//*************************************************************************************************************************************************************************

//Perform State tasks here

// Send hold command to all sub modules
SubModulesCollection.NotifyStateChanged(ePMLCommand_Hold);

IF NOT SubModulesCollection.AllInRequestedState(ePMLState_Held) THEN
	RETURN;
END_IF

StateComplete();
END_METHOD

//! @summary This method contains code which will execute when this PackML module is in the <b>Idle</b> state
METHOD PROTECTED Idle

(*! <description> <b>The base implementation of this method is empty. User must override this method to provide functionality.</b>
<table> 
	<tr>
		<th> Previous State </th>
		<th> Transition In </th>
		<th> Transition Out </th>
		<th> Next State  </th> 
	</tr>
	<tr>
		<td> Resetting </td>
		<td> State Complete <i>(Resetting)</i></td> 
		<td> Start Command </td>
		<td> Starting </td> 
	</tr>
</table>
This method is called as required by <c>StateControl()</c>
</description> 

*)
//*************************************************************************************************************************************************************************

//If you are about to write application specific code, note that any such code should exist within the "Application" directory using a Function Block that 'EXTENDS' this base Function Block!

//This particular method's functionality can be overriden in the extended block by creating a method of the same name, with desired functionality therein

//If the functionality of this base module is to be retained, but more functionality is desired, the extended method can contain a SUPER^.ThisMethodName(); call, which will call this code

//*************************************************************************************************************************************************************************
END_METHOD

//! @summary Basic module initialization logic
METHOD PROTECTED Initialize : BOOL;
//! @description This method is called by <c>CyclicLogic()</c> as required
//This method may get called several times while waiting for subunits/components to init

//so it makes sense to break it up into a state machine

CASE InitialiseStates OF
  init:
    CreateEvents();
    InitialiseStates := CountSubModules;

  CountSubModules:
    // Figure out how many Submodules were instantiated - they should be from 1 to X and not skip any indices.
    NumberOfSubModules := SubModulesCollection.Count;
	//SubModulesCollection.SetPMLSubModuleInfoActive(PMLSubModuleInfo);
    InitialiseStates := SetSizeOfArrays;
	
  SetSizeOfArrays:
    // Initialize subunit overview used by state machine
//    PMLSubModuleInfoRef.ArraySize := SIZEOF(PMLSubModuleInfo);
//    PMLSubModuleInfoRef.NoOfSubUnits := NumberOfSubModules;
//    PMLSubModuleInfoRef.pArray := ADR(PMLSubModuleInfo);
    InitialiseStates := WaitForInitializeComplete;
	
  WaitForInitializeComplete:
	SubModulesCollection.CyclicLogic();
	componentsCollection.CyclicLogic();

    IF SubModulesCollection.InitialisedAll AND componentsCollection.InitialisedAll THEN
      InitialiseStates := init;
      Initialize := TRUE;
    END_IF
END_CASE
END_METHOD

PROPERTY PUBLIC LogModeChanges : BOOL
GET
LogModeChanges := ModeManager.LogModeChanges;
END_GET
SET
ModeManager.LogModeChanges := LogModeChanges;
END_SET
END_PROPERTY

//! @summary Enable/Disable logging of state changes
PROPERTY LogStateChanges : BOOL
GET
LogStateChanges := _LogStateChanges;
END_GET
SET
_LogStateChanges := LogStateChanges;
END_SET
END_PROPERTY

//! @summary Sets the requested PackML Mode
PROPERTY ModeCommand : DINT
GET
ModeCommand := ModeManager.CommandedMode;
END_GET
SET
VAR
	i : UDINT;
END_VAR
//IF ModeCommand <> _CommandedMode THEN
//    _CommandedMode                    := ModeCommand;
//    PackMLBaseModule_HMI.Command.Mode := ModeCommand;
	
//    //Notify external controllers that state has changed	
//    FOR i := 1 TO Parameters_PackML_Base.MAX_NO_OF_EXTERNAL_CONTROLLERS DO
//        IF ipExternalControllers[i] <> 0 THEN
//            ipExternalControllers[i].ModeChanged(_CommandedMode);
//        END_IF
//    END_FOR
    
//    //ModeChangeRequested := TRUE;
//END_IF
END_SET
END_PROPERTY

//! @summary Handles mode change requests for this module and all submodules
METHOD PRIVATE FINAL ModeControl
VAR
    i : UDINT;
END_VAR

//! @description This method is called cyclically by <c>CyclicLogic()</c>
(*
//On startup, Mode is invalid, set it to production

IF _CurrentMode = E_PMLUnitMode.ePMLUnitMode_Invalid THEN
    ModeChangeRequested := TRUE;
    _CommandedMode      := Parameters_PackML_Base.UNIT_MODE_DEFAULT;

    //Notify external controllers that state has changed	
    FOR i := 1 TO Parameters_PackML_Base.MAX_NO_OF_EXTERNAL_CONTROLLERS DO
        IF ipExternalControllers[i] <> 0 THEN
            ipExternalControllers[i].ModeChanged(_CommandedMode);
        END_IF
    END_FOR

    LastModeCommand := _CommandedMode;
    

    //If mode is valid and the command has changed, attempt to change modes
ELSIF _CommandedMode <> LastModeCommand THEN
    ModeChangeRequested               := TRUE;
    PackMLBaseModule_HMI.Command.Mode := _CommandedMode;

    //Notify external controllers that state has changed	
    FOR i := 1 TO Parameters_PackML_Base.MAX_NO_OF_EXTERNAL_CONTROLLERS DO
        IF ipExternalControllers[i] <> 0 THEN
            ipExternalControllers[i].ModeChanged(_CommandedMode);
        END_IF
    END_FOR

    LastModeCommand := _CommandedMode;
END_IF

IF ModeChangeRequested THEN
    //Handles mode changes based on ModeCommand and the state transition rules defined in the pre-defined protected modes or custom modes
    ModeManager(bExecute     := TRUE,
                eModeCommand := _CommandedMode,
                eState       := _CurrentState,
                eModeStatus  => _CurrentMode);

    IF ModeManager.bDone THEN
        IF PackMLAlarms[E_PackMLBase_Alarms.ModeCommandInvalid].bRaised THEN
            PackMLAlarms[E_PackMLBase_Alarms.ModeCommandInvalid].Clear(0, 0);
        END_IF

        //If PackML mode has changed
        IF ModeManager.eModeStatus <> LastMode THEN
            LastMode                := ModeManager.eModeStatus;
            SequenceState           := 0;
            DescendantSequenceState := 0;

            //If state change logging is not suppressed
            IF _LogModeChanges THEN
                PMLModeLogger(Alarms := PackMLAlarms, ModulePrefix := _Name, Mode := ModeManager.eModeStatus);
            END_IF

            // Change SubModules
            FOR i := 1 TO NumberOfSubModules DO
                ipSubModules[i].ModeCommand := ModeManager.eModeStatus; //Call the SetMode loop of the subunits 
            END_FOR
        END_IF

        // Reset mode control command
        ModeManager(bExecute := FALSE);
        ModeChangeRequested := FALSE;
    ELSIF ModeManager.bError THEN
        IF ReachedInitialDefaultStateAndMode THEN
            IF NOT PackMLAlarms[E_PackMLBase_Alarms.ModeCommandInvalid].bRaised THEN
                PackMLAlarms[E_PackMLBase_Alarms.ModeCommandInvalid].Raise(0);
            END_IF
        END_IF

        // Reset mode control command
        ModeManager(bExecute := FALSE);
        ModeChangeRequested := FALSE;
    END_IF
END_IF
*)
END_METHOD

//! @summary Get/Set the name of this module
PROPERTY Name : STRING
GET
Name := _Name;
END_GET
SET
_Name := Name;
END_SET
END_PROPERTY

//! @summary TODO: does this do anything?
PROPERTY ParentResponseDefinitions : ARRAY[0..4] OF E_AlarmResponse
GET
ParentResponseDefinitions[TcEventSeverity.Verbose]  := _ParentFaultResponseDefinitions[TcEventSeverity.Verbose];
ParentResponseDefinitions[TcEventSeverity.Info]     := _ParentFaultResponseDefinitions[TcEventSeverity.Info];
ParentResponseDefinitions[TcEventSeverity.Warning]  := _ParentFaultResponseDefinitions[TcEventSeverity.Warning];
ParentResponseDefinitions[TcEventSeverity.Error]    := _ParentFaultResponseDefinitions[TcEventSeverity.Error];
ParentResponseDefinitions[TcEventSeverity.Critical] := _ParentFaultResponseDefinitions[TcEventSeverity.Critical];
END_GET
SET
_ParentFaultResponseDefinitions[TcEventSeverity.Verbose]  := ParentResponseDefinitions[TcEventSeverity.Verbose];
_ParentFaultResponseDefinitions[TcEventSeverity.Info]     := ParentResponseDefinitions[TcEventSeverity.Info];
_ParentFaultResponseDefinitions[TcEventSeverity.Warning]  := ParentResponseDefinitions[TcEventSeverity.Warning];
_ParentFaultResponseDefinitions[TcEventSeverity.Error]    := ParentResponseDefinitions[TcEventSeverity.Error];
_ParentFaultResponseDefinitions[TcEventSeverity.Critical] := ParentResponseDefinitions[TcEventSeverity.Critical];
END_SET
END_PROPERTY

//! @summary Raises an alarm and passes string arguments as parameters for extra fault context/info
METHOD PROTECTED RaiseAlarmWithStrings
VAR_IN_OUT
    Alarm : FB_TcAlarm; //! Alarm to be raised
END_VAR

VAR_INPUT
    String_1 : STRING; //! First string parameter (The Name of this component will be applied first automatically)
    String_2 : STRING; //! Second string parameter
END_VAR
F_RaiseAlarmWithStringParameters(Alarm    := Alarm,
                                 String_1 := Name,
                                 String_2 := String_1,
                                 String_3 := String_2);
END_METHOD

METHOD FINAL RegisterExternalController : BOOL
VAR_INPUT
    Controller : I_PackML_ExternalController;
END_VAR

VAR
    i : UDINT;
END_VAR
IF NOT ExternalControllersCollection.AddController(Controller) THEN
	RETURN;
END_IF

Controller.Control         := THIS^;
RegisterExternalController := TRUE;
END_METHOD

//! @summary This method contains code which will execute when this PackML module is in the <b>Resetting</b> state
METHOD PROTECTED Resetting
VAR
    i               : UDINT;
    SubModulesReady : BOOL := TRUE;
	Module : I_PackML_BaseModule;
END_VAR

(*! <description> <b>Note:</b> The <i>Reset</i> command can also be thought of as an <i>enable</i> depite the ambiguity in the naming of the <i>Clearing</i> state.
<table> 
	<tr>
		<th> Previous State </th>
		<th> Transition In </th>
		<th> Transition Out </th>
		<th> Next State  </th> 
	</tr>
	<tr>
		<td> Stopped<b>-or-</b>Completed </td>
		<td> Reset Command </td> 
		<td> State Complete </td>
		<td> Idle </td> 
	</tr>
</table>
This method is called as required by <c>StateControl()</c>
</description> 

*)
//*************************************************************************************************************************************************************************

//If you are about to write application specific code, note that any such code should exist within the "Application" directory using a Function Block that 'EXTENDS' this base Function Block!

//This particular method's functionality can be overriden in the extended block by creating a method of the same name, with desired functionality therein

//If the functionality of this base module is to be retained, but more functionality is desired, the extended method can contain a SUPER^.ThisMethodName(); call, which will call this code

//*************************************************************************************************************************************************************************

//Perform State tasks here

// Send clear/reset command to all sub modules

//As long as this module is in the "Resetting" state, it will attempt to get all modules to Idle by sending abort, clear, and reset commands as appropriate to its children until they do


//FOR i := 1 TO NumberOfSubModules DO
//    IF ipSubModules[i].CurrentState = ePMLState_Stopped OR ipSubModules[i].CurrentState = ePMLState_Complete THEN
//        ipSubModules[i].StateCommand := ePMLCommand_Reset;
//    ELSIF ipSubModules[i].CurrentState = ePMLState_Aborted THEN
//        ipSubModules[i].StateCommand := ePMLCommand_Clear;
//    ELSIF ipSubModules[i].CurrentState = ePMLState_Clearing OR ipSubModules[i].CurrentState = ePMLState_Stopping OR ipSubModules[i].CurrentState = ePMLState_Resetting OR
//          ipSubModules[i].CurrentState = ePMLState_Idle THEN
//        ;
//    ELSE
//        ipSubModules[i].StateCommand := ePMLCommand_Abort;
//    END_IF
//END_FOR

SubModulesCollection.StateReset();

IF NOT SubModulesCollection.AllInRequestedState(ePMLState_Idle) THEN
	RETURN;
END_IF

StateComplete();
END_METHOD

//! @summary This method contains code which will execute when this PackML module is in the <b>Starting</b> state
METHOD PROTECTED Starting
VAR
    i               : UDINT;
    SubModulesReady : BOOL := TRUE;
END_VAR

(*! <description><b></b><table> 
	<tr>
		<th> Previous State </th>
		<th> Transition In </th>
		<th> Transition Out </th>
		<th> Next State  </th> 
	</tr>
	<tr>
		<td> Idle </td>
		<td> Start Command </td> 
		<td> State Complete </td>
		<td> Execute </td> 
	</tr>
</table>
This method is called as required by <c>StateControl()</c>
</description> 

*)
//*************************************************************************************************************************************************************************

//If you are about to write application specific code, note that any such code should exist within the "Application" directory using a Function Block that 'EXTENDS' this base Function Block!

//This particular method's functionality can be overriden in the extended block by creating a method of the same name, with desired functionality therein

//If the functionality of this base module is to be retained, but more functionality is desired, the extended method can contain a SUPER^.ThisMethodName(); call, which will call this code

//*************************************************************************************************************************************************************************

//Perform State tasks here

// Send start command to all sub modules
SubModulesCollection.NotifyStateChanged(ePMLCommand_Start);

IF NOT SubModulesCollection.AllInRequestedState(ePMLState_Execute) THEN
	RETURN;
END_IF

StateComplete();
END_METHOD

METHOD PRIVATE StartUpStateTransition
//On startup, state is invalid, set it to default
IF _CurrentState = E_PMLState.ePMLState_Undefined AND ModeManager.CurrentMode <> E_PMLUnitMode.ePMLUnitMode_Invalid THEN
    _CommandedState := Parameters_PackML_Base.UNIT_STATE_DEFAULT;
END_IF
END_METHOD

//! @summary Sets the requested PackML state
PROPERTY StateCommand : Tc3_PackML_V2.E_PMLCommand
GET
StateCommand := _CommandedState;
END_GET
SET
VAR
	i : UDINT;
END_VAR
IF ModeManager.CurrentMode <> E_PMLUnitMode.ePMLUnitMode_Invalid AND _CurrentState <> E_PMLState.ePMLState_Undefined THEN

    _CommandedState                    := StateCommand;
    PackMLBaseModule_HMI.Command.State := StateCommand;	
	ExternalControllersCollection.NotifyStateChanged (_CommandedState);

END_IF
END_SET
END_PROPERTY

//! @summary Signals to the state manager FB when a state has completed
METHOD PROTECTED StateComplete

//! @description This method is called by any of the transition state's logic methods (<c>...<b>ing()</b></c>) as required
//*************************************************************************************************************************************************************************

//If you are about to write application specific code, note that any such code should exist within the "Application" directory using a Function Block that 'EXTENDS' this base Function Block!

//This particular method's functionality can be overriden in the extended block by creating a method of the same name, with desired functionality therein

//If the functionality of this base module is to be retained, but more functionality is desired, the extended method can contain a SUPER^.ThisMethodName(); call, which will call this code

//*************************************************************************************************************************************************************************
StateMachine.M_StateComplete();
END_METHOD

//! @summary Calls PackML state manager and corresponding methods according to current module state
METHOD PRIVATE FINAL StateControl
//! @description This method is called cyclically by <c>CyclicLogic()</c>
VAR
    i : UDINT;
END_VAR
StartUpStateTransition();

//Call PackML state machine	
StateMachine(
  eMode := ModeManager.CurrentMode,
  eCommand := _CommandedState,
  eState => _CurrentState
);

//If PackML state has changed
IF _CurrentState <> PrevState THEN
  PrevState := _CurrentState;
  PackMLBaseModule_HMI.Command.State := _CommandedState;

  //Notify external controllers that state has changed
  ExternalControllersCollection.NotifyStateChanged (_CommandedState);

  InitialiseStates := init;
END_IF

IF ReachedInitialDefaultStateAndMode THEN
  //Log appropriate state changes
  PMLStateLogger(
    Alarms := PackMLAlarms,
    ModulePrefix := _Name,
    State := _CurrentState,
    LogAllChanges := _LogStateChanges
  );
END_IF

// Call appropriate method depending on current PackML state
CASE _CurrentState OF
  E_PMLState.ePMLState_Undefined:
    Undefined();
  E_PMLState.ePMLState_Clearing:
    Clearing();
  E_PMLState.ePMLState_Stopped:
    Stopped();
  E_PMLState.ePMLState_Starting:
    Starting();
  E_PMLState.ePMLState_Idle:
    Idle();
  E_PMLState.ePMLState_Suspended:
    Suspended();
  E_PMLState.ePMLState_Execute:
    Execute();
  E_PMLState.ePMLState_Stopping:
    Stopping();
  E_PMLState.ePMLState_Aborting:
    Aborting();
  E_PMLState.ePMLState_Aborted:
    Aborted();
  E_PMLState.ePMLState_Holding:
    Holding();
  E_PMLState.ePMLState_Held:
    Held();
  E_PMLState.ePMLState_Unholding:
    Unholding();
  E_PMLState.ePMLState_Suspending:
    Suspending();
  E_PMLState.ePMLState_Unsuspending:
    Unsuspending();
  E_PMLState.ePMLState_Resetting:
    Resetting();
  E_PMLState.ePMLState_Completing:
    Completing();
  E_PMLState.ePMLState_Complete:
    Complete();
END_CASE
END_METHOD

//! @summary Provides fault reaction logic where the module state is driven to the <b>Stopping</b> state at the next available opportunity
METHOD PROTECTED StopControlled

(*! <description> No error is thrown by this fault reaction.
	<b> TODO: Needs implementation </b> </description>*)

//! @description This method is called by <c>ComponentMonitor()</c> or <c>SubModuleMonitor()</c> as required
ChangeState(E_PMLCommand.ePMLCommand_Stop);
END_METHOD

//! @summary Provides fault reaction logic where the module state is driven to the <b>Stopping</b> state immediately
METHOD PROTECTED StopImmediate

//! @description No error is thrown by this fault reaction.

//! @description This method is called by <c>ComponentMonitor()</c> or <c>SubModuleMonitor()</c> as required
ChangeState(E_PMLCommand.ePMLCommand_Stop);
END_METHOD

//! @summary This method contains code which will execute when this PackML module is in the <b>Stopped</b> state
METHOD PROTECTED Stopped

(*! <description> <b>The base implementation of this method is empty. User must override this method to provide functionality.</b>
<table> 
	<tr>
		<th> Previous State </th>
		<th> Transition In </th>
		<th> Transition Out </th>
		<th> Next State  </th> 
	</tr>
	<tr>
		<td> Stopping<b>-or-</b>Clearing </td>
		<td> State Complete <i>(Stopping<b>-or-</b>Clearing)</i></td> 
		<td> Reset Command </td>
		<td> Resetting </td> 
	</tr>
</table>
This method is called as required by <c>StateControl()</c>
</description> 

*)
//*************************************************************************************************************************************************************************

//If you are about to write application specific code, note that any such code should exist within the "Application" directory using a Function Block that 'EXTENDS' this base Function Block!

//This particular method's functionality can be overriden in the extended block by creating a method of the same name, with desired functionality therein

//If the functionality of this base module is to be retained, but more functionality is desired, the extended method can contain a SUPER^.ThisMethodName(); call, which will call this code

//*************************************************************************************************************************************************************************
END_METHOD

//! @summary This method contains code which will execute when this PackML module is in the <b>Stopping</b> state
METHOD PROTECTED Stopping
VAR
    i               : UDINT;
    SubModulesReady : BOOL := TRUE;
END_VAR

(*! <description><b></b><table> 
	<tr>
		<th> Previous State </th>
		<th> Transition In </th>
		<th> Transition Out </th>
		<th> Next State  </th> 
	</tr>
	<tr>
		<td> <b>ANY<i>except</i></b>Stopped<b>-or-</b>Clearing<b>-or-</b>Aborted<b>-or-</b>Aborting</td>
		<td> Stop Command </td> 
		<td> State Complete </td>
		<td> Stopped </td> 
	</tr>
</table>
This method is called as required by <c>StateControl()</c>
</description> 

*)
//*************************************************************************************************************************************************************************

//If you are about to write application specific code, note that any such code should exist within the "Application" directory using a Function Block that 'EXTENDS' this base Function Block!

//This particular method's functionality can be overriden in the extended block by creating a method of the same name, with desired functionality therein

//If the functionality of this base module is to be retained, but more functionality is desired, the extended method can contain a SUPER^.ThisMethodName(); call, which will call this code

//*************************************************************************************************************************************************************************

//Perform State tasks here

// Send stop command to all sub modules
SubModulesCollection.NotifyStateChanged(ePMLCommand_Stop);

IF SubModulesCollection.AllInRequestedState(ePMLState_Stopped) 
	OR SubModulesCollection.AllInRequestedState(ePMLState_Aborted) THEN
	
	StateComplete();
END_IF
END_METHOD

//! @summary This method monitors <b>submodules</b> within this PackML module and initiates fault responses as required
METHOD PROTECTED SubModuleMonitor : BOOL
VAR
    AlarmResponses : ARRAY[0..4] OF E_AlarmResponse; //Temporary response array	
    i              : UDINT;
END_VAR

//! @description This method is called cyclically by <c>CyclicLogic()</c>
//SubModulesCollection.GetAlarmResponse(_CurrentState);

FOR i := 1 TO NumberOfSubModules DO
    IF _CurrentState <> E_PMLState.ePMLState_Aborted AND _CurrentState <> E_PMLState.ePMLState_Aborting AND _CurrentState <> E_PMLState.ePMLState_Clearing AND
       _CurrentState <> E_PMLState.ePMLState_Stopped AND _CurrentState <> E_PMLState.ePMLState_Stopping THEN
        AlarmResponses := ipSubModules[i].ParentResponseDefinitions;
        
        CASE AlarmResponses[ipSubModules[i].CurrentAlarmSeverity] OF
            E_AlarmResponse.Abort_ImmediateError:
                AbortImmediateError(ipSubModules[i].Name, TRUE);

            E_AlarmResponse.Abort_Immediate:
                AbortImmediate();

            E_AlarmResponse.Stop_Immediate:
                StopImmediate();

            E_AlarmResponse.Stop_Controlled:
                StopControlled();

            E_AlarmResponse.Hold_Immediate:
                HoldImmediate();

            E_AlarmResponse.Suspend_Immediate:
                SuspendImmediate();

            E_AlarmResponse.Suspend_Controlled:
                SuspendControlled();

            E_AlarmResponse.NoResponse:
                ;
        END_CASE
    ELSIF _CurrentState = E_PMLState.ePMLState_Stopped OR _CurrentState = E_PMLState.ePMLState_Stopping THEN
        AlarmResponses := ipSubModules[i].ParentResponseDefinitions;
        CASE AlarmResponses[ipSubModules[i].CurrentAlarmSeverity] OF
            E_AlarmResponse.Abort_ImmediateError:
                AbortImmediateError(ipSubModules[i].Name, TRUE);

            E_AlarmResponse.Abort_Immediate:
                AbortImmediate();

            E_AlarmResponse.NoResponse:
                ;
        END_CASE
    END_IF
END_FOR
END_METHOD

//! @summary Provides fault reaction logic where the module state is driven to the <b>Suspending</b> state at the next available opportunity
METHOD PROTECTED SuspendControlled

(*! <description> No error is thrown by this fault reaction.
	<b> TODO: Needs implementation </b> </description>*)

//! @description This method is called by <c>ComponentMonitor()</c> or <c>SubModuleMonitor()</c> as required
ChangeState(E_PMLCommand.ePMLCommand_Suspend);
END_METHOD

//! @summary This method contains code which will execute when this PackML module is in the <b>Suspended</b> state
METHOD PROTECTED Suspended

(*! <description> <b>The base implementation of this method is empty. User must override this method to provide functionality.</b>
<table> 
	<tr>
		<th> Previous State </th>
		<th> Transition In </th>
		<th> Transition Out </th>
		<th> Next State  </th> 
	</tr>
	<tr>
		<td> Suspending </td>
		<td> State Complete <i>(Suspending)</i></td> 
		<td> Unsuspend Command </td>
		<td> Unsuspending </td> 
	</tr>
</table>
This method is called as required by <c>StateControl()</c>
</description> 

*)
//*************************************************************************************************************************************************************************

//If you are about to write application specific code, note that any such code should exist within the "Application" directory using a Function Block that 'EXTENDS' this base Function Block!

//This particular method's functionality can be overriden in the extended block by creating a method of the same name, with desired functionality therein

//If the functionality of this base module is to be retained, but more functionality is desired, the extended method can contain a SUPER^.ThisMethodName(); call, which will call this code

//*************************************************************************************************************************************************************************
END_METHOD

//! @summary Provides fault reaction logic where the module state is driven to the <b>Suspending</b> state immediately
METHOD PROTECTED SuspendImmediate

(*! <description> No error is thrown by this fault reaction.
	<b> TODO: Needs implementation </b> </description>*)

//! @description This method is called by <c>ComponentMonitor()</c> or <c>SubModuleMonitor()</c> as required
ChangeState(E_PMLCommand.ePMLCommand_Suspend);
END_METHOD

//! @summary This method contains code which will execute when this PackML module is in the <b>Suspending</b> state
METHOD PROTECTED Suspending
VAR
    i               : UDINT;
    SubModulesReady : BOOL := TRUE;
END_VAR

(*! <description><b>Note:</b> The <i>Suspend</i> command is intended to be initiated by automatic detection of upstream/downstream jams, etc. It is meant to be distinct from a <i>Hold</i> in that <i>Hold</i> should be commanded by an operator.  Both <i>Hold</i>and<i>Suspend</i> result in a <i>paused</i> state which should allow resumption of the <b>Execute</b> state. 
<table> 
	<tr>
		<th> Previous State </th>
		<th> Transition In </th>
		<th> Transition Out </th>
		<th> Next State  </th> 
	</tr>
	<tr>
		<td> Execute </td>
		<td> Suspend Command </td> 
		<td> State Complete </td>
		<td> Suspended </td> 
	</tr>
</table>
This method is called as required by <c>StateControl()</c>
</description> 

*)
//*************************************************************************************************************************************************************************

//If you are about to write application specific code, note that any such code should exist within the "Application" directory using a Function Block that 'EXTENDS' this base Function Block!

//This particular method's functionality can be overriden in the extended block by creating a method of the same name, with desired functionality therein

//If the functionality of this base module is to be retained, but more functionality is desired, the extended method can contain a SUPER^.ThisMethodName(); call, which will call this code

//*************************************************************************************************************************************************************************

//Perform State tasks here

// Send suspend command to all sub modules
SubModulesCollection.NotifyStateChanged(ePMLCommand_Suspend);

IF NOT SubModulesCollection.AllInRequestedState(ePMLState_Suspended) THEN
	RETURN;
END_IF

StateComplete();
END_METHOD

//! @summary This method contains code which will execute when this PackML module is in a state which is not defined by the PackML standard
METHOD PROTECTED Undefined

(*! <description> <b>The base implementation of this method is empty. User must override this method to provide functionality.
<i>This state should not be reached under normal circumstances.</i></b>
This method is called as required by <c>StateControl()</c>
</description> 

*)
//*************************************************************************************************************************************************************************

//If you are about to write application specific code, note that any such code should exist within the "Application" directory using a Function Block that 'EXTENDS' this base Function Block!

//This particular method's functionality can be overriden in the extended block by creating a method of the same name, with desired functionality therein

//If the functionality of this base module is to be retained, but more functionality is desired, the extended method can contain a SUPER^.ThisMethodName(); call, which will call this code

//*************************************************************************************************************************************************************************
END_METHOD

//! @summary This method contains code which will execute when this PackML module is in the <b>Unholding</b> state
METHOD PROTECTED Unholding
VAR
    i               : UDINT;
    SubModulesReady : BOOL := TRUE;
END_VAR

(*! <description><b></b><table> 
	<tr>
		<th> Previous State </th>
		<th> Transition In </th>
		<th> Transition Out </th>
		<th> Next State  </th> 
	</tr>
	<tr>
		<td> Held </td>
		<td> Unhold Command </td> 
		<td> State Complete </td>
		<td> Execute </td> 
	</tr>
</table>
This method is called as required by <c>StateControl()</c>
</description> 

*)
//*************************************************************************************************************************************************************************

//If you are about to write application specific code, note that any such code should exist within the "Application" directory using a Function Block that 'EXTENDS' this base Function Block!

//This particular method's functionality can be overriden in the extended block by creating a method of the same name, with desired functionality therein

//If the functionality of this base module is to be retained, but more functionality is desired, the extended method can contain a SUPER^.ThisMethodName(); call, which will call this code

//*************************************************************************************************************************************************************************

//Perform State tasks here

// Send unhold command to all sub modules
SubModulesCollection.NotifyStateChanged(ePMLCommand_Unhold);

IF NOT SubModulesCollection.AllInRequestedState(ePMLState_Execute) THEN
	RETURN;
END_IF

StateComplete();
END_METHOD

//! @summary This method contains code which will execute when this PackML module is in the <b>Unsuspending</b> state
METHOD PROTECTED Unsuspending
VAR
    i               : UDINT;
    SubModulesReady : BOOL := TRUE;
END_VAR

(*! <description><b></b><table> 
	<tr>
		<th> Previous State </th>
		<th> Transition In </th>
		<th> Transition Out </th>
		<th> Next State  </th> 
	</tr>
	<tr>
		<td> Suspended </td>
		<td> Unsuspend Command </td> 
		<td> State Complete </td>
		<td> Execute </td> 
	</tr>
</table>
This method is called as required by <c>StateControl()</c>
</description> 

*)
//*************************************************************************************************************************************************************************

//If you are about to write application specific code, note that any such code should exist within the "Application" directory using a Function Block that 'EXTENDS' this base Function Block!

//This particular method's functionality can be overriden in the extended block by creating a method of the same name, with desired functionality therein

//If the functionality of this base module is to be retained, but more functionality is desired, the extended method can contain a SUPER^.ThisMethodName(); call, which will call this code

//*************************************************************************************************************************************************************************

//Perform State tasks here

// Send unsuspend command to all sub modules
SubModulesCollection.NotifyStateChanged(ePMLCommand_Unsuspend);

IF NOT SubModulesCollection.AllInRequestedState(ePMLState_Execute) THEN
	RETURN;
END_IF

StateComplete();
END_METHOD

END_FUNCTION_BLOCK

// ---- Intecre/ModeManager/T_ModeManager.TcPOU
FUNCTION_BLOCK T_ModeManager IMPLEMENTS I_ModeManager
VAR
  _state : I_StateModule;
  _LogModeChanges : BOOL := TRUE;
  _CurrentMode, PrevCurrentMode : E_PMLUnitMode; //Current UnitMode of the module	
  _CommandedMode, PrevCommandedMode : E_PMLUnitMode; //Current Commanded UnitMode of the module

  PackModeManager : PML_UnitModeManager;
  CustomModes : PML_UnitModeConfig;
  PMLModeLogger : FB_PackML_ModeLogger;

  _ModeNames : ARRAY[0..31] OF STRING; // ('Production','Maintenance', 'Manual');

  CurrentStrategy : I_PackMode := ProductionMode;
  ProductionMode : I_PackMode;
  MaintenanceMode : I_PackMode;
  ManualMode : I_PackMode;
  CustomPackModes : ARRAY[0..15] OF I_PackMode; // mobject ?
END_VAR

METHOD AddCustomPackMode : BOOL
VAR_INPUT
  index : UINT;
  newPackMode : I_PackMode;
END_VAR
custompackmodes[index] := newPackMode;
END_METHOD

METHOD AddPackModes : BOOL
VAR_INPUT
  prodMode : I_PackMode;
  maintMode : I_PackMode;
  manMode : I_PackMode;
END_VAR
ProductionMode := prodMode;
MaintenanceMode := maintMode;
ManualMode := manMode;
END_METHOD

METHOD PUBLIC AddStateModule
VAR_INPUT
  stateModule : I_StateModule;
END_VAR
_state := stateModule;
END_METHOD

METHOD PUBLIC ChangeMode
VAR_INPUT
  Mode : E_PMLUnitMode;
END_VAR
IF Mode <> _CommandedMode THEN
    _CommandedMode := Mode;
END_IF
END_METHOD

PROPERTY PUBLIC CommandedMode : E_PMLUnitMode
GET
CommandedMode := _CommandedMode;
END_GET
END_PROPERTY

PROPERTY CurrentMode : E_PMLUnitMode
GET
CurrentMode := _CurrentMode;
END_GET
END_PROPERTY

METHOD PUBLIC CyclicLogic
VAR_INPUT
END_VAR
ModeControl();
END_METHOD

METHOD FB_init : BOOL
VAR_INPUT
	bInitRetains : BOOL; // if TRUE, the retain variables are initialized (warm start / cold start)
	bInCopyCode : BOOL;  // if TRUE, the instance afterwards gets moved into the copy code (online change)
  	stateModule : I_StateModule;
END_VAR
_state := stateModule;
END_METHOD

PROPERTY PUBLIC LogModeChanges : BOOL
GET
LogModeChanges := _LogModeChanges;
END_GET
SET
_LogModeChanges := LogModeChanges;
END_SET
END_PROPERTY

METHOD PRIVATE ModeChange
//Handles mode changes based on ModeCommand and the state transition rules defined in the pre-defined protected modes or custom modes
PackModeManager(
  bExecute := ModeChangeRequested,
  eModeCommand := _CommandedMode,
  eState := _state.CurrentState,
  eModeStatus => _CurrentMode
);

IF PackModeManager.bError THEN
  _CommandedMode := PrevCommandedMode;

ELSIF PackModeManager.bDone THEN
  PrevCurrentMode := _CurrentMode;
  PrevCommandedMode := _CommandedMode;
  SetCurrentStrategy(_CurrentMode);
END_IF

//TODO how to get loggin and alarms out from here?
END_METHOD

PROPERTY ModeChangeRequested : BOOL
GET
ModeChangeRequested := _CommandedMode <> PrevCommandedMode;
END_GET
END_PROPERTY

METHOD PRIVATE ModeControl //Final ?
VAR
END_VAR
StartUpModeChange();
ModeChange();
END_METHOD

PROPERTY PUBLIC  ModeNames : REFERENCE TO ARRAY[0..31] OF STRING
GET
ModeNames REF= _ModeNames;
END_GET
END_PROPERTY

METHOD PRIVATE SetCurrentStrategy
VAR_INPUT
	CurrentMode : E_PMLUnitMode;
END_VAR
CASE CurrentMode OF
	E_PMLUnitMode.ePMLUnitMode_Maintenance :
		CurrentStrategy := MaintenanceMode;
	E_PMLUnitMode.ePMLUnitMode_Manual :
		CurrentStrategy := ManualMode;	
	E_PMLUnitMode.ePMLUnitMode_Production :
		CurrentStrategy := ProductionMode;
	ELSE
		;//?
END_CASE
END_METHOD

METHOD PRIVATE StartUpModeChange
//On startup, Mode is invalid, set it to production
IF _CurrentMode = E_PMLUnitMode.ePMLUnitMode_Invalid THEN
  _CommandedMode := Parameters_PackML_Base.UNIT_MODE_DEFAULT;
END_IF
END_METHOD

END_FUNCTION_BLOCK

// ---- FB_PackML_ModeLogger.TcPOU
//! @summary This FB raises events corresponding to <b>mode</b> changes within the parent PackML module
FUNCTION_BLOCK FB_PackML_ModeLogger
VAR_IN_OUT
    Alarms : ARRAY[1..48] OF FB_TcAlarm; //! Array of alarms for Core PackML events that exist in any PackML enabled module
END_VAR

VAR_INPUT
    ModulePrefix : STRING; //! Prefix String for any  <TODO> Remove this? </TODO>
    Mode         : DINT;   //! Current mode of the module
END_VAR

VAR
    LastMode : DINT;
END_VAR

IF Mode <> LastMode THEN
    CASE Mode OF
        E_PMLUnitMode.ePMLUnitMode_Invalid:
            Alarms[E_PackMLBase_Alarms.ModeInvalidEnter].Raise(0);
        E_PMLUnitMode.ePMLUnitMode_Production:
            Alarms[E_PackMLBase_Alarms.ModeProductionEnter].Raise(0);
        E_PMLUnitMode.ePMLUnitMode_Maintenance:
            Alarms[E_PackMLBase_Alarms.ModeMaintenanceEnter].Raise(0);
        E_PMLUnitMode.ePMLUnitMode_Manual:
            Alarms[E_PackMLBase_Alarms.ModeManualEnter].Raise(0);
    END_CASE

    CASE LastMode OF
        E_PMLUnitMode.ePMLUnitMode_Invalid:
            Alarms[E_PackMLBase_Alarms.ModeInvalidEnter].Clear(0, 0);
        E_PMLUnitMode.ePMLUnitMode_Production:
            Alarms[E_PackMLBase_Alarms.ModeProductionEnter].Clear(0, 0);
        E_PMLUnitMode.ePMLUnitMode_Maintenance:
            Alarms[E_PackMLBase_Alarms.ModeMaintenanceEnter].Clear(0, 0);
        E_PMLUnitMode.ePMLUnitMode_Manual:
            Alarms[E_PackMLBase_Alarms.ModeManualEnter].Clear(0, 0);
    END_CASE

    LastMode := Mode;
END_IF

(*! <description> The current mode is compared against the mode during the last call.  The corresponding events are raised/cleared as the mode is changed.
<b>This FB is called from FB_PMLModuleBase.ModeControl.  Further calls are not necessary.</b></description>*)

END_FUNCTION_BLOCK

// ---- Intecre/Collections/T_ComponentsCollection.TcPOU
FUNCTION_BLOCK T_ComponentsCollection EXTENDS T_NamedBase IMPLEMENTS I_ComponentsCollection
VAR
	baseCollection : T_CollectionBase;
END_VAR

METHOD PUBLIC AddComponent : BOOL
VAR_INPUT
  newComponent : I_ComponentBase;
END_VAR
IF newComponent = 0 THEN
	LogError( 'Cannot AddComponent invalid ref' );
	RETURN;
END_IF

AddComponent := baseCollection.AddItem( newItem := CastToBase(newComponent) );
END_METHOD

METHOD PUBLIC AllowHMIControl
VAR
	i : UDINT;
	Component : I_ComponentBase;
END_VAR
IF Count = 0 THEN
    RETURN;
END_IF

WHILE i < Count 
		AND_THEN TryGetComponent(i, component => Component) DO
		
    Component.AllowHMIControl();
    i := i + 1;
END_WHILE
END_METHOD

PROPERTY PUBLIC AnyError : BOOL
GET
VAR
  i : UDINT;
  Component : I_ComponentBase;
END_VAR
IF Count = 0 THEN
    RETURN;
END_IF

FOR i := 0 TO Count - 1 DO

    IF NOT TryGetComponent(i, component => Component) THEN
        RETURN;
    END_IF
		
	IF Component.Error THEN
		AnyError := TRUE;
		RETURN;
	END_IF

END_FOR
END_GET
END_PROPERTY

METHOD PUBLIC BlockHMIControl
VAR
	i : UDINT;
	Component : I_ComponentBase;
END_VAR
IF Count = 0 THEN
    RETURN;
END_IF

WHILE i < Count 
		AND_THEN TryGetComponent(i, component => Component) DO
		
    Component.BlockHMIControl();
    i := i + 1;
END_WHILE
END_METHOD

METHOD PRIVATE CastToBase : I_InterfaceBase
VAR_INPUT
	Component : I_ComponentBase;
END_VAR
__QUERYINTERFACE(Component, CastToBase);
END_METHOD

METHOD PRIVATE CastToType : I_ComponentBase
VAR_INPUT
	Base : I_InterfaceBase;
END_VAR
__QUERYINTERFACE(Base, CastToType);
END_METHOD

METHOD PUBLIC ClearGroup // clears the group down
baseCollection.ClearGroup();
END_METHOD

PROPERTY Count : UDINT
GET
Count := baseCollection.Count;
END_GET
END_PROPERTY

METHOD CyclicLogic
VAR
  i : UDINT;
  Component : I_ComponentBase;
END_VAR
IF Count = 0 THEN
    RETURN;
END_IF

WHILE i < Count 
		AND_THEN TryGetComponent(i, component => Component) DO
		
    Component.CyclicLogic();
    i := i + 1;
END_WHILE
END_METHOD

PROPERTY PUBLIC InitialisedAll : BOOL
GET
VAR
  i : UDINT;
  Component : I_ComponentBase;
 END_VAR
IF Count = 0 THEN
    InitialisedAll := TRUE;
    RETURN;
END_IF

WHILE i < Count 
		AND_THEN TryGetComponent(i, component => Component) DO
		
    IF NOT Component.InitComplete THEN
		RETURN;
	END_IF
	
    i := i + 1;
END_WHILE

InitialisedAll := TRUE;
END_GET
END_PROPERTY

METHOD PUBLIC Reset
VAR
	i : UDINT;
	Component : I_ComponentBase;
END_VAR
IF Count = 0 THEN
    RETURN;
END_IF

WHILE i < Count 
		AND_THEN TryGetComponent(i, component => Component) DO
		
    IF Component.Error THEN
		Component.Reset();
	END_IF
	
    i := i + 1;
END_WHILE
END_METHOD

METHOD TryGetComponent: BOOL
VAR_INPUT
	index : UDINT;
END_VAR
VAR_OUTPUT
	component : I_ComponentBase;
END_VAR
VAR
	baseItem : I_InterfaceBase;
END_VAR
baseCollection.TryGetItem(index, item => baseItem);
component := CastToType(baseItem);

IF component = 0 THEN
	LogError( 'Cannot TryGetComponent  component = 0' );
	RETURN;
END_IF 

TryGetComponent := component <> 0;
END_METHOD

END_FUNCTION_BLOCK

// ---- Intecre/Collections/T_CollectionBase.TcPOU
FUNCTION_BLOCK T_CollectionBase EXTENDS T_NamedBase
VAR
    _items : ARRAY[0..(COLLECTION_MAX_SIZE-1)] OF I_InterfaceBase;
    _cnt : UDINT;
END_VAR
VAR CONSTANT
    COLLECTION_MAX_SIZE : UDINT := Parameters_PackML_Base.COLLECTION_MAX_SIZE;
END_VAR

METHOD PRIVATE addInSpareSlot : BOOL
VAR_INPUT
	Item : I_InterfaceBase;
END_VAR
IF Count >= COLLECTION_MAX_SIZE THEN
	LogError('cannot addInSpareSlot : no space.');
	RETURN;
END_IF
	
_items[Count] := Item;
Count := Count + 1;
addInSpareSlot := TRUE;
END_METHOD

METHOD INTERNAL AddItem : BOOL
VAR_INPUT
  newItem : I_InterfaceBase;
END_VAR
IF newItem = 0 THEN
	LogError( 'Cannot AddComponent invalid ref' );
	RETURN;
END_IF

IF HasItem( Item := newItem ) THEN
	LogWarning( 'Component already in collection.' );
	RETURN;
END_IF

AddItem := addInSpareSlot( Item := newItem );
END_METHOD

METHOD ClearGroup // clears the group down
MEMSET(ADR(_items), 0 , SIZEOF(_items));
_cnt := 0;
LogDebug('ClearGroup() called.');
END_METHOD

PROPERTY Count : UDINT
GET
Count := _cnt;
END_GET
SET // PRIVATE
_cnt := Count;
END_SET
END_PROPERTY

METHOD PRIVATE HasItem : BOOL
VAR_INPUT
	Item : I_InterfaceBase;
END_VAR
VAR 
	i : UDINT;
END_VAR
IF Count >= COLLECTION_MAX_SIZE THEN
	LogWarning('Count Exceed Collection Max Size');
	RETURN;
END_IF

FOR i := 0 TO Count DO
	
	IF _items[i] = 0 THEN
		EXIT; // exit for loop
	END_IF
	
	IF _items[i] = Item THEN
		HasItem := TRUE;
		RETURN;
		
	END_IF
	
END_FOR
END_METHOD

METHOD INTERNAL TryGetItem: BOOL
VAR_INPUT
	index : UDINT;
END_VAR
VAR_OUTPUT
	item : I_InterfaceBase;
END_VAR
IF index > (COLLECTION_MAX_SIZE-1) THEN
	LogError( 'cannot GetDrive, index out of bounds' );
	RETURN;
END_IF

IF index > Count THEN
	LogError( 'cannot GetDrive, index > (Count - 1) ' );
	RETURN;
END_IF

item := _items[index];
TryGetItem := item <> 0;
END_METHOD

END_FUNCTION_BLOCK

// ---- Intecre/Collections/T_SubModuleCollection.TcPOU
FUNCTION_BLOCK T_SubModuleCollection EXTENDS T_NamedBase IMPLEMENTS I_SubModuleCollection
VAR
	baseCollection : T_CollectionBase;
END_VAR

METHOD PUBLIC AddModule : BOOL
VAR_INPUT
  newModule : I_PackML_BaseModule;
END_VAR
IF newModule = 0 THEN
	LogError( 'Cannot AddModule invalid ref' );
	RETURN;
END_IF

AddModule := baseCollection.AddItem( newItem := CastToBase(newModule) );
END_METHOD

METHOD PUBLIC AllInRequestedState : BOOL
VAR_INPUT
	State : Tc3_PackML_V2.E_PMLState;
END_VAR
VAR
	i : UDINT;
	Module : I_PackML_BaseModule;
END_VAR
IF Count = 0 THEN
	AllInRequestedState := TRUE;
	RETURN;
END_IF

WHILE i < Count 
		AND_THEN TryGetModule(i, Module => Module) DO
		
    IF Module.CurrentState <> State THEN
		RETURN;
	END_IF
	
    i := i + 1;
END_WHILE

AllInRequestedState := TRUE;
END_METHOD

PROPERTY AnyError : BOOL
GET
VAR
  i : UDINT;
  Module : I_PackML_BaseModule;
 END_VAR
IF Count = 0 THEN
    RETURN;
END_IF

FOR i := 0 TO Count - 1 DO

    IF NOT TryGetModule(i, Module => Module) THEN
        RETURN;
    END_IF
		
	IF Module.Error THEN
		AnyError := TRUE;
		RETURN;
	END_IF

END_FOR
END_GET
END_PROPERTY

METHOD PUBLIC AnyInRequestedState : BOOL
VAR_INPUT
	State : Tc3_PackML_V2.E_PMLState;
END_VAR
VAR_OUTPUT
	Module : I_PackML_BaseModule;	
END_VAR
VAR
	i : UDINT;
END_VAR
WHILE i < Count 
		AND_THEN TryGetModule(i, Module => Module) DO
		
    IF Module.CurrentState = State THEN
		AnyInRequestedState := TRUE;
		RETURN;
	END_IF
	
    i := i + 1;
END_WHILE
END_METHOD

METHOD PRIVATE CastToBase : I_InterfaceBase
VAR_INPUT
	Module : I_PackML_BaseModule;
END_VAR
__QUERYINTERFACE(Module, CastToBase);
END_METHOD

METHOD PRIVATE CastToType : I_PackML_BaseModule
VAR_INPUT
	Base : I_InterfaceBase;
END_VAR
__QUERYINTERFACE(Base, CastToType);
END_METHOD

METHOD PUBLIC ClearGroup // clears the group down
baseCollection.ClearGroup();
END_METHOD

PROPERTY Count : UDINT
GET
Count := baseCollection.Count;
END_GET
END_PROPERTY

METHOD CyclicLogic
VAR
  i : UDINT;
  Module : I_PackML_BaseModule;
END_VAR
WHILE i < Count 
		AND_THEN TryGetModule(i, Module => Module) DO
		
    Module.CyclicLogic();
    i := i + 1;
END_WHILE
END_METHOD

PROPERTY PUBLIC InitialisedAll : BOOL
GET
VAR
  i : UDINT;
  Module : I_PackML_BaseModule;
 END_VAR
IF Count = 0 THEN
	InitialisedAll := TRUE;
  RETURN;
END_IF

WHILE i < Count 
		AND_THEN TryGetModule(i, Module => Module) DO
		
	IF NOT Module.InitComplete THEN
		RETURN;
	END_IF
    i := i + 1;
END_WHILE

InitialisedAll := TRUE;
END_GET
END_PROPERTY

METHOD PUBLIC NotifyModeChanged
VAR_INPUT
    Mode : E_PMLUnitMode;
END_VAR
VAR
	i : UDINT;
	Module : I_PackML_BaseModule;
END_VAR
WHILE i < Count 
		AND_THEN TryGetModule(i, Module => Module) DO
		
	Module.ChangeMode(Mode);
    i := i + 1;
END_WHILE
END_METHOD

METHOD PUBLIC NotifyStateChanged
VAR_INPUT
	CommandedState : Tc3_PackML_V2.E_PMLCommand;
END_VAR
VAR
	i : UDINT;
	Module : I_PackML_BaseModule;
END_VAR
WHILE i < Count 
		AND_THEN TryGetModule(i, Module => Module) DO
		
	Module.ChangeState(CommandedState);
    i := i + 1;
END_WHILE
END_METHOD

METHOD PUBLIC StateReset
VAR
	i : UDINT;
	Module : I_PackML_BaseModule;
END_VAR
IF Count = 0 THEN
	RETURN;
END_IF


WHILE i < Count 
		AND_THEN TryGetModule(i, Module => Module) DO
	
	IF Module.CurrentState = ePMLState_Stopped OR Module.CurrentState = ePMLState_Complete THEN
		Module.ChangeState (ePMLCommand_Reset);
	ELSIF Module.CurrentState = ePMLState_Aborted THEN
		Module.ChangeState (ePMLCommand_Clear);
	ELSIF Module.CurrentState = ePMLState_Clearing OR Module.CurrentState = ePMLState_Stopping OR Module.CurrentState = ePMLState_Resetting OR
		 Module.CurrentState = ePMLState_Idle THEN
		;
	ELSE
		Module.ChangeState(ePMLCommand_Abort);
	END_IF
		
	
    i := i + 1;
	
END_WHILE
END_METHOD

METHOD TryGetModule: BOOL
VAR_INPUT
	index : UDINT;
END_VAR
VAR_OUTPUT
	Module : I_PackML_BaseModule;
END_VAR
VAR
	baseItem : I_InterfaceBase;
END_VAR
baseCollection.TryGetItem(index, item => baseItem);
Module := CastToType(baseItem);

IF Module = 0 THEN
	LogError( 'Cannot TryGetModule  Module = 0' );
	RETURN;
END_IF 

TryGetModule := Module <> 0;
END_METHOD

END_FUNCTION_BLOCK

// ---- Intecre/Collections/T_ExternalControllerCollection.TcPOU
FUNCTION_BLOCK T_ExternalControllerCollection EXTENDS T_NamedBase;
VAR
	baseCollection : T_CollectionBase;
END_VAR

METHOD PUBLIC AddController : BOOL
VAR_INPUT
  newController : I_PackML_ExternalController;
END_VAR
IF newController = 0 THEN
	LogError( 'Cannot AddController invalid ref' );
	RETURN;
END_IF

AddController := baseCollection.AddItem( newItem := CastToBase(newController) );
END_METHOD

METHOD PRIVATE CastToBase : I_InterfaceBase
VAR_INPUT
	Controller : I_PackML_ExternalController;
END_VAR
__QUERYINTERFACE(Controller, CastToBase);
END_METHOD

METHOD PRIVATE CastToType : I_PackML_ExternalController
VAR_INPUT
	Base : I_InterfaceBase;
END_VAR
__QUERYINTERFACE(Base, CastToType);
END_METHOD

METHOD PUBLIC ClearGroup // clears the group down
baseCollection.ClearGroup();
END_METHOD

PROPERTY Count : UDINT
GET
Count := baseCollection.Count;
END_GET
END_PROPERTY

METHOD PUBLIC NotifyModeChanged
VAR_INPUT
    Mode : E_PMLUnitMode;
END_VAR
VAR
	i : UDINT;
	Controller : I_PackML_ExternalController;
END_VAR
WHILE i < Count 
		AND_THEN TryGetController(i, Controller => Controller) DO
		
    Controller.ModeChanged(Mode);
    i := i + 1;
END_WHILE
END_METHOD

METHOD PUBLIC NotifyStateChanged
VAR_INPUT
	CommandedState : Tc3_PackML_V2.E_PMLCommand;
END_VAR
VAR
	i : UDINT;
	Controller : I_PackML_ExternalController;
END_VAR
WHILE i < Count 
		AND_THEN TryGetController(i, Controller => Controller) DO
		
    Controller.StateChanged(CommandedState);
    i := i + 1;
END_WHILE
END_METHOD

METHOD TryGetController: BOOL
VAR_INPUT
	index : UDINT;
END_VAR
VAR_OUTPUT
	Controller : I_PackML_ExternalController;
END_VAR
VAR
	baseItem : I_InterfaceBase;
END_VAR
baseCollection.TryGetItem(index, item => baseItem);
Controller := CastToType(baseItem);

IF Controller = 0 THEN
	LogError( 'Cannot TryGetController  Controller = 0' );
	RETURN;
END_IF 

TryGetController := Controller <> 0;
END_METHOD

END_FUNCTION_BLOCK

// ---- Intecre/Collections/T_BaseAlarms.TcPOU
FUNCTION_BLOCK T_BaseAlarms EXTENDS T_NamedBase
VAR
	alarms : ARRAY[E_BaseAlarms.InitReferenceEvent..E_BaseAlarms.InvalidInterface] OF FB_TcAlarm;
END_VAR
VAR CONSTANT
	USE_DEFAULT_TIMESTAMP : ULINT := 0; // If default then it will use system time, else it will use timestamp 
  //https://infosys.beckhoff.com/english.php?content=../content/1033/tc3_eventlogger/5050505739.html&id=8432917619912920197
END_VAR

PROPERTY AlarmsArray : REFERENCE TO ARRAY[E_BaseAlarms.InitReferenceEvent..E_BaseAlarms.InvalidInterface] OF FB_TcAlarm
GET
AlarmsArray REF= alarms;
END_GET
END_PROPERTY

METHOD ClearAlarmIfRaised
VAR_INPUT
	alarm : E_BaseAlarms;
	resetConfirmation : BOOL;
END_VAR
IF NOT alarms[alarm].bRaised THEN
	RETURN;
END_IF

alarms[alarm].Clear(USE_DEFAULT_TIMESTAMP,resetConfirmation);
END_METHOD

METHOD RaiseAlarmWithStringParameters
VAR_INPUT
	alarm : E_BaseAlarms;

